LIN {X 0,Y 418.273,Z 271.104,A -85,B 0,C 180,E1 -10135.819,E2 -10135.819} C_VEL
LIN {X 0,Y 422.663,Z 288.535,A -85,B 0,C 180,E1 -10138.973,E2 -10138.973} C_VEL
LIN {X 0,Y 424.828,Z 297.383,A -85,B 0,C 180,E1 -10140.52,E2 -10140.52} C_VEL
LIN {X 0,Y 424.797,Z 302.116,A -85,B 0,C 180,E1 -10141.265,E2 -10141.265} C_VEL
LIN {X 0,Y 423.732,Z 315.882,A -85,B 0,C 180,E1 -10143.326,E2 -10143.326} C_VEL
LIN {X 0,Y 429.33,Z 349.112,A -85,B 0,C 180,E1 -10144.378,E2 -10144.378} C_VEL
LIN {X 0,Y 426.147,Z 475.897,A -85,B 0,C 180,E1 -10146.942,E2 -10146.942} C_VEL
LIN {X 0,Y 425.571,Z 491.648,A -85,B 0,C 180,E1 -10147.359,E2 -10147.359} C_VEL
LIN {X 0,Y 424.744,Z 507.01,A -85,B 0,C 180,E1 -10147.955,E2 -10147.955} C_VEL
LIN {X 0,Y 423.794,Z 521.926,A -85,B 0,C 180,E1 -10148.732,E2 -10148.732} C_VEL
LIN {X 0,Y 422.751,Z 536.416,A -85,B 0,C 180,E1 -10149.696,E2 -10149.696} C_VEL
LIN {X 0,Y 421.703,Z 549.683,A -85,B 0,C 180,E1 -10150.784,E2 -10150.784} C_VEL
LIN {X 0,Y 420.781,Z 561.783,A -85,B 0,C 180,E1 -10151.981,E2 -10151.981} C_VEL
LIN {X 0,Y 419.884,Z 572.417,A -85,B 0,C 180,E1 -10153.22,E2 -10153.22} C_VEL
LIN {X 0,Y 419.045,Z 583.025,A -85,B 0,C 180,E1 -10154.685,E2 -10154.685} C_VEL
LIN {X 0,Y 418.331,Z 593.403,A -85,B 0,C 180,E1 -10156.398,E2 -10156.398} C_VEL
LIN {X 0,Y 417.855,Z 601.99,A -85,B 0,C 180,E1 -10158.111,E2 -10158.111} C_VEL
LIN {X 0,Y 417.459,Z 609.054,A -85,B 0,C 180,E1 -10159.82,E2 -10159.82} C_VEL
LIN {X 0,Y 417.247,Z 615.562,A -85,B 0,C 180,E1 -10161.77,E2 -10161.77} C_VEL
LIN {X 0,Y 417.123,Z 620.649,A -85,B 0,C 180,E1 -10163.763,E2 -10163.763} C_VEL
LIN {X 0,Y 417.095,Z 623.363,A -85,B 0,C 180,E1 -10165.169,E2 -10165.169} C_VEL
LIN {X 0,Y 417.171,Z 625.963,A -85,B 0,C 180,E1 -10167.104,E2 -10167.104} C_VEL
LIN {X 0,Y 417.117,Z 627.235,A -85,B 0,C 180,E1 -10169.036,E2 -10169.036} C_VEL
LIN {X 0,Y 417.106,Z 627.238,A -85,B 0,C 180,E1 -10170.967,E2 -10170.967} C_VEL
LIN {X 0,Y 417.167,Z 625.984,A -85,B 0,C 180,E1 -10172.898,E2 -10172.898} C_VEL
LIN {X 0,Y 417.113,Z 623.451,A -85,B 0,C 180,E1 -10174.834,E2 -10174.834} C_VEL
LIN {X 0,Y 417.146,Z 619.609,A -85,B 0,C 180,E1 -10176.774,E2 -10176.774} C_VEL
LIN {X 0,Y 417.27,Z 614.36,A -85,B 0,C 180,E1 -10178.72,E2 -10178.72} C_VEL
LIN {X 0,Y 417.572,Z 607.571,A -85,B 0,C 180,E1 -10180.67,E2 -10180.67} C_VEL
LIN {X 0,Y 417.913,Z 600.256,A -85,B 0,C 180,E1 -10182.382,E2 -10182.382} C_VEL
LIN {X 0,Y 418.554,Z 591.444,A -85,B 0,C 180,E1 -10184.093,E2 -10184.093} C_VEL
LIN {X 0,Y 419.389,Z 580.845,A -85,B 0,C 180,E1 -10185.803,E2 -10185.803} C_VEL
LIN {X 0,Y 420.33,Z 569.042,A -85,B 0,C 180,E1 -10187.391,E2 -10187.391} C_VEL
LIN {X 0,Y 421.444,Z 557.196,A -85,B 0,C 180,E1 -10188.725,E2 -10188.725} C_VEL
LIN {X 0,Y 422.596,Z 544.432,A -85,B 0,C 180,E1 -10189.934,E2 -10189.934} C_VEL
LIN {X 0,Y 423.78,Z 530.617,A -85,B 0,C 180,E1 -10191.017,E2 -10191.017} C_VEL
LIN {X 0,Y 424.991,Z 515.84,A -85,B 0,C 180,E1 -10191.956,E2 -10191.956} C_VEL
LIN {X 0,Y 426.146,Z 500.139,A -85,B 0,C 180,E1 -10192.733,E2 -10192.733} C_VEL
LIN {X 0,Y 427.209,Z 483.991,A -85,B 0,C 180,E1 -10193.32,E2 -10193.32} C_VEL
LIN {X 0,Y 428.073,Z 463.838,A -85,B 0,C 180,E1 -10193.815,E2 -10193.815} C_VEL
LIN {X 0,Y 431.123,Z 384.555,A -85,B 0,C 180,E1 -10195.656,E2 -10195.656} C_VEL
LIN {X 0,Y 432.678,Z 349.283,A -85,B 0,C 180,E1 -10196.531,E2 -10196.531} C_VEL
LIN {X 0,Y 430.547,Z 332.583,A -85,B 0,C 180,E1 -10197.238,E2 -10197.238} C_VEL
LIN {X 0,Y 427.37,Z 315.726,A -85,B 0,C 180,E1 -10198.1,E2 -10198.1} C_VEL
LIN {X 0,Y 425.847,Z 308.551,A -85,B 0,C 180,E1 -10198.531,E2 -10198.531} C_VEL
LIN {X 0,Y 426.669,Z 302.236,A -85,B 0,C 180,E1 -10199.615,E2 -10199.615} C_VEL
LIN {X 0,Y 425.498,Z 295.343,A -85,B 0,C 180,E1 -10201.076,E2 -10201.076} C_VEL
LIN {X 0,Y 423.264,Z 286.408,A -85,B 0,C 180,E1 -10203.227,E2 -10203.227} C_VEL
LIN {X 0,Y 420.793,Z 278.456,A -85,B 0,C 180,E1 -10205.474,E2 -10205.474} C_VEL
LIN {X 0,Y 418.246,Z 271.014,A -85,B 0,C 180,E1 -10208.054,E2 -10208.054} C_VEL
LIN {X 0,Y 418.229,Z 271.016,A -85,B 0,C 180,E1 -10210.948,E2 -10210.948} C_VEL
LIN {X 0,Y 418.216,Z 271.017,A -85,B 0,C 180,E1 -10213.73,E2 -10213.73} C_VEL
LIN {X 0,Y 418.216,Z 271.016,A -85,B 0,C 180,E1 -10216.449,E2 -10216.449} C_VEL
LIN {X 0,Y 418.229,Z 271.015,A -85,B 0,C 180,E1 -10219.131,E2 -10219.131} C_VEL
LIN {X 0,Y 418.233,Z 271.014,A -85,B 0,C 180,E1 -10222.167,E2 -10222.167} C_VEL
LIN {X 0,Y 418.272,Z 271.011,A -85,B 0,C 180,E1 -10225.42,E2 -10225.42} C_VEL
LIN {X 0,Y 418.236,Z 271.089,A -85,B 0,C 180,E1 -10227.898,E2 -10227.898} C_VEL
LIN {X 0,Y 420.645,Z 278.367,A -85,B 0,C 180,E1 -10230.749,E2 -10230.749} C_VEL
LIN {X 0,Y 420.932,Z 279.274,A -85,B 0,C 180,E1 -10231.015,E2 -10231.015} C_VEL
LIN {X 0,Y 426.506,Z 288.448,A -85,B 0,C 180,E1 -10232.033,E2 -10232.033} C_VEL
LIN {X 0,Y 431.738,Z 298.009,A -85,B 0,C 180,E1 -10232.929,E2 -10232.929} C_VEL
LIN {X 0,Y 434.186,Z 303.111,A -85,B 0,C 180,E1 -10233.341,E2 -10233.341} C_VEL
LIN {X 0,Y 430.286,Z 382.983,A -85,B 0,C 180,E1 -10235.321,E2 -10235.321} C_VEL
LIN {X 0,Y 428.073,Z 441.208,A -85,B 0,C 180,E1 -10236.698,E2 -10236.698} C_VEL
LIN {X 0,Y 427.292,Z 456.973,A -85,B 0,C 180,E1 -10237.262,E2 -10237.262} C_VEL
LIN {X 0,Y 426.378,Z 472.657,A -85,B 0,C 180,E1 -10238.039,E2 -10238.039} C_VEL
LIN {X 0,Y 425.436,Z 486.789,A -85,B 0,C 180,E1 -10238.942,E2 -10238.942} C_VEL
LIN {X 0,Y 424.349,Z 500.509,A -85,B 0,C 180,E1 -10240.026,E2 -10240.026} C_VEL
LIN {X 0,Y 423.148,Z 512.964,A -85,B 0,C 180,E1 -10241.212,E2 -10241.212} C_VEL
LIN {X 0,Y 422.024,Z 524.671,A -85,B 0,C 180,E1 -10242.556,E2 -10242.556} C_VEL
LIN {X 0,Y 421.067,Z 535.277,A -85,B 0,C 180,E1 -10244.013,E2 -10244.013} C_VEL
LIN {X 0,Y 419.97,Z 545.744,A -85,B 0,C 180,E1 -10245.734,E2 -10245.734} C_VEL
LIN {X 0,Y 419.183,Z 554.155,A -85,B 0,C 180,E1 -10247.41,E2 -10247.41} C_VEL
LIN {X 0,Y 418.633,Z 560.313,A -85,B 0,C 180,E1 -10248.868,E2 -10248.868} C_VEL
LIN {X 0,Y 418.092,Z 567.004,A -85,B 0,C 180,E1 -10250.81,E2 -10250.81} C_VEL
LIN {X 0,Y 417.678,Z 572.295,A -85,B 0,C 180,E1 -10252.798,E2 -10252.798} C_VEL
LIN {X 0,Y 417.441,Z 575.139,A -85,B 0,C 180,E1 -10254.202,E2 -10254.202} C_VEL
LIN {X 0,Y 417.373,Z 577.965,A -85,B 0,C 180,E1 -10256.137,E2 -10256.137} C_VEL
LIN {X 0,Y 417.231,Z 579.565,A -85,B 0,C 180,E1 -10258.069,E2 -10258.069} C_VEL
LIN {X 0,Y 417.12,Z 579.956,A -85,B 0,C 180,E1 -10259.999,E2 -10259.999} C_VEL
LIN {X 0,Y 417.179,Z 579.128,A -85,B 0,C 180,E1 -10261.93,E2 -10261.93} C_VEL
LIN {X 0,Y 417.263,Z 577.05,A -85,B 0,C 180,E1 -10263.862,E2 -10263.862} C_VEL
LIN {X 0,Y 417.383,Z 573.711,A -85,B 0,C 180,E1 -10265.798,E2 -10265.798} C_VEL
LIN {X 0,Y 417.568,Z 569.044,A -85,B 0,C 180,E1 -10267.737,E2 -10267.737} C_VEL
LIN {X 0,Y 417.904,Z 562.933,A -85,B 0,C 180,E1 -10269.681,E2 -10269.681} C_VEL
LIN {X 0,Y 418.46,Z 555.198,A -85,B 0,C 180,E1 -10271.626,E2 -10271.626} C_VEL
LIN {X 0,Y 419.056,Z 546.461,A -85,B 0,C 180,E1 -10273.411,E2 -10273.411} C_VEL
LIN {X 0,Y 419.798,Z 536.838,A -85,B 0,C 180,E1 -10275.039,E2 -10275.039} C_VEL
LIN {X 0,Y 420.628,Z 526.543,A -85,B 0,C 180,E1 -10276.501,E2 -10276.501} C_VEL
LIN {X 0,Y 421.633,Z 514.5,A -85,B 0,C 180,E1 -10277.934,E2 -10277.934} C_VEL
LIN {X 0,Y 422.485,Z 501.996,A -85,B 0,C 180,E1 -10279.179,E2 -10279.179} C_VEL
LIN {X 0,Y 423.522,Z 488.72,A -85,B 0,C 180,E1 -10280.266,E2 -10280.266} C_VEL
LIN {X 0,Y 424.403,Z 474.164,A -85,B 0,C 180,E1 -10281.237,E2 -10281.237} C_VEL
LIN {X 0,Y 425.216,Z 459.835,A -85,B 0,C 180,E1 -10281.985,E2 -10281.985} C_VEL
LIN {X 0,Y 425.821,Z 444.87,A -85,B 0,C 180,E1 -10282.579,E2 -10282.579} C_VEL
LIN {X 0,Y 426.282,Z 429.156,A -85,B 0,C 180,E1 -10283.007,E2 -10283.007} C_VEL
LIN {X 0,Y 429.565,Z 298.762,A -85,B 0,C 180,E1 -10285.643,E2 -10285.643} C_VEL
LIN {X 0,Y 420.488,Z 276.554,A -85,B 0,C 180,E1 -10286.661,E2 -10286.661} C_VEL
LIN {X 0,Y 418.28,Z 271.31,A -85,B 0,C 180,E1 -10286.912,E2 -10286.912} C_VEL
LIN {X 0,Y 418.245,Z 271.009,A -85,B 0,C 180,E1 -10286.98,E2 -10286.98} C_VEL
LIN {X 0,Y 418.243,Z 271.013,A -85,B 0,C 180,E1 -10290.271,E2 -10290.271} C_VEL
LIN {X 0,Y 418.249,Z 271.012,A -85,B 0,C 180,E1 -10293.676,E2 -10293.676} C_VEL
LIN {X 0,Y 418.238,Z 271.009,A -85,B 0,C 180,E1 -10297.223,E2 -10297.223} C_VEL
LIN {X 0,Y 418.228,Z 271.015,A -85,B 0,C 180,E1 -10299.683,E2 -10299.683} C_VEL
LIN {X 0,Y 418.222,Z 271.012,A -85,B 0,C 180,E1 -10302.319,E2 -10302.319} C_VEL
LIN {X 0,Y 418.234,Z 271.009,A -85,B 0,C 180,E1 -10305.107,E2 -10305.107} C_VEL
LIN {X 0,Y 418.238,Z 271.015,A -85,B 0,C 180,E1 -10307.765,E2 -10307.765} C_VEL
LIN {X 0,Y 418.243,Z 271.008,A -85,B 0,C 180,E1 -10310.619,E2 -10310.619} C_VEL
LIN {X 0,Y 418.239,Z 271.013,A -85,B 0,C 180,E1 -10313.974,E2 -10313.974} C_VEL
LIN {X 0,Y 418.253,Z 271.008,A -85,B 0,C 180,E1 -10317.155,E2 -10317.155} C_VEL
LIN {X 0,Y 418.257,Z 271.006,A -85,B 0,C 180,E1 -10320.836,E2 -10320.836} C_VEL
LIN {X 0,Y 418.233,Z 271.012,A -85,B 0,C 180,E1 -10324.092,E2 -10324.092} C_VEL
LIN {X 0,Y 418.227,Z 271.012,A -85,B 0,C 180,E1 -10327.262,E2 -10327.262} C_VEL
LIN {X 0,Y 418.277,Z 271.004,A -85,B 0,C 180,E1 -10330.363,E2 -10330.363} C_VEL
LIN {X 0,Y 418.31,Z 271.004,A -85,B 0,C 180,E1 -10333.403,E2 -10333.403} C_VEL
LIN {X 0,Y 418.34,Z 270.996,A -85,B 0,C 180,E1 -10336.998,E2 -10336.998} C_VEL
LIN {X 0,Y 418.315,Z 270.999,A -85,B 0,C 180,E1 -10339.744,E2 -10339.744} C_VEL
LIN {X 0,Y 417.662,Z 271.081,A -85,B 0,C 180,E1 -10340.548,E2 -10340.548} C_VEL
LIN {X 0,Y 414.856,Z 271.434,A -85,B 0,C 180,E1 -10341.857,E2 -10341.857} C_VEL
LIN {X 0,Y 412.502,Z 271.724,A -85,B 0,C 180,E1 -10342.914,E2 -10342.914} C_VEL
LIN {X 0,Y 411.52,Z 271.851,A -85,B 0,C 180,E1 -10343.73,E2 -10343.73} C_VEL
LIN {X 0,Y 411.456,Z 271.854,A -85,B 0,C 180,E1 -10344.006,E2 -10344.006} C_VEL
LIN {X 0,Y 411.502,Z 271.849,A -85,B 0,C 180,E1 -10348.041,E2 -10348.041} C_VEL
LIN {X 0,Y 411.633,Z 271.833,A -85,B 0,C 180,E1 -10349.999,E2 -10349.999} C_VEL
LIN {X 0,Y 411.449,Z 271.855,A -85,B 0,C 180,E1 -10352.936,E2 -10352.936} C_VEL
LIN {X 0,Y 411.448,Z 271.855,A -85,B 0,C 180,E1 -10356.866,E2 -10356.866} C_VEL
LIN {X 0,Y 411.344,Z 271.868,A -85,B 0,C 180,E1 -10358.844,E2 -10358.844} C_VEL
LIN {X 0,Y 411.273,Z 271.879,A -85,B 0,C 180,E1 -10361.832,E2 -10361.832} C_VEL
LIN {X 0,Y 411.249,Z 271.88,A -85,B 0,C 180,E1 -10364.852,E2 -10364.852} C_VEL
LIN {X 0,Y 411.241,Z 271.882,A -85,B 0,C 180,E1 -10367.914,E2 -10367.914} C_VEL
LIN {X 0,Y 411.184,Z 271.89,A -85,B 0,C 180,E1 -10371.033,E2 -10371.033} C_VEL
LIN {X 0,Y 411.213,Z 271.884,A -85,B 0,C 180,E1 -10374.214,E2 -10374.214} C_VEL
LIN {X 0,Y 411.246,Z 271.886,A -85,B 0,C 180,E1 -10377.477,E2 -10377.477} C_VEL
LIN {X 0,Y 411.176,Z 271.89,A -85,B 0,C 180,E1 -10380.847,E2 -10380.847} C_VEL
LIN {X 0,Y 411.192,Z 271.886,A -85,B 0,C 180,E1 -10384.333,E2 -10384.333} C_VEL
LIN {X 0,Y 411.186,Z 271.888,A -85,B 0,C 180,E1 -10387.972,E2 -10387.972} C_VEL
LIN {X 0,Y 411.151,Z 271.898,A -85,B 0,C 180,E1 -10391.228,E2 -10391.228} C_VEL
LIN {X 0,Y 411.167,Z 271.889,A -85,B 0,C 180,E1 -10394.489,E2 -10394.489} C_VEL
LIN {X 0,Y 411.164,Z 271.889,A -85,B 0,C 180,E1 -10398.194,E2 -10398.194} C_VEL
LIN {X 0,Y 411.202,Z 271.887,A -85,B 0,C 180,E1 -10400.776,E2 -10400.776} C_VEL
LIN {X 0,Y 411.183,Z 271.887,A -85,B 0,C 180,E1 -10404.471,E2 -10404.471} C_VEL
LIN {X 0,Y 411.192,Z 271.889,A -85,B 0,C 180,E1 -10406.873,E2 -10406.873} C_VEL
LIN {X 0,Y 411.218,Z 271.884,A -85,B 0,C 180,E1 -10410.644,E2 -10410.644} C_VEL
LIN {X 0,Y 411.223,Z 271.884,A -85,B 0,C 180,E1 -10413.619,E2 -10413.619} C_VEL
LIN {X 0,Y 411.182,Z 271.891,A -85,B 0,C 180,E1 -10416.852,E2 -10416.852} C_VEL
LIN {X 0,Y 411.2,Z 271.885,A -85,B 0,C 180,E1 -10420.051,E2 -10420.051} C_VEL
LIN {X 0,Y 411.249,Z 271.886,A -85,B 0,C 180,E1 -10423.131,E2 -10423.131} C_VEL
LIN {X 0,Y 411.291,Z 271.878,A -85,B 0,C 180,E1 -10426.896,E2 -10426.896} C_VEL
LIN {X 0,Y 411.279,Z 271.875,A -85,B 0,C 180,E1 -10430.162,E2 -10430.162} C_VEL
LIN {X 0,Y 411.438,Z 271.862,A -85,B 0,C 180,E1 -10433.133,E2 -10433.133} C_VEL
LIN {X 0,Y 411.294,Z 271.88,A -85,B 0,C 180,E1 -10435.1,E2 -10435.1} C_VEL
LIN {X 0,Y 411.501,Z 271.847,A -85,B 0,C 180,E1 -10438.043,E2 -10438.043} C_VEL
LIN {X 0,Y 411.628,Z 271.832,A -85,B 0,C 180,E1 -10440.001,E2 -10440.001} C_VEL
LIN {X 0,Y 411.444,Z 271.861,A -85,B 0,C 180,E1 -10442.938,E2 -10442.938} C_VEL
LIN {X 0,Y 411.446,Z 271.86,A -85,B 0,C 180,E1 -10446.868,E2 -10446.868} C_VEL
LIN {X 0,Y 411.342,Z 271.873,A -85,B 0,C 180,E1 -10448.846,E2 -10448.846} C_VEL
LIN {X 0,Y 411.273,Z 271.876,A -85,B 0,C 180,E1 -10451.834,E2 -10451.834} C_VEL
LIN {X 0,Y 411.248,Z 271.885,A -85,B 0,C 180,E1 -10454.854,E2 -10454.854} C_VEL
LIN {X 0,Y 411.241,Z 271.88,A -85,B 0,C 180,E1 -10457.916,E2 -10457.916} C_VEL
LIN {X 0,Y 411.186,Z 271.892,A -85,B 0,C 180,E1 -10461.035,E2 -10461.035} C_VEL
LIN {X 0,Y 411.209,Z 271.885,A -85,B 0,C 180,E1 -10464.217,E2 -10464.217} C_VEL
LIN {X 0,Y 411.249,Z 271.88,A -85,B 0,C 180,E1 -10467.479,E2 -10467.479} C_VEL
LIN {X 0,Y 411.18,Z 271.895,A -85,B 0,C 180,E1 -10470.849,E2 -10470.849} C_VEL
LIN {X 0,Y 411.197,Z 271.887,A -85,B 0,C 180,E1 -10474.335,E2 -10474.335} C_VEL
LIN {X 0,Y 411.184,Z 271.887,A -85,B 0,C 180,E1 -10477.975,E2 -10477.975} C_VEL
LIN {X 0,Y 411.155,Z 271.893,A -85,B 0,C 180,E1 -10481.23,E2 -10481.23} C_VEL
LIN {X 0,Y 411.168,Z 271.893,A -85,B 0,C 180,E1 -10484.492,E2 -10484.492} C_VEL
LIN {X 0,Y 411.171,Z 271.89,A -85,B 0,C 180,E1 -10488.196,E2 -10488.196} C_VEL
LIN {X 0,Y 411.213,Z 271.89,A -85,B 0,C 180,E1 -10490.778,E2 -10490.778} C_VEL
LIN {X 0,Y 411.192,Z 271.888,A -85,B 0,C 180,E1 -10494.473,E2 -10494.473} C_VEL
LIN {X 0,Y 411.24,Z 272.041,A -85,B 0,C 180,E1 -10495.468,E2 -10495.468} C_VEL
LIN {X 0,Y 415.179,Z 287.627,A -85,B 0,C 180,E1 -10498.35,E2 -10498.35} C_VEL
LIN {X 0,Y 418.118,Z 300.046,A -85,B 0,C 180,E1 -10500.553,E2 -10500.553} C_VEL
LIN {X 0,Y 416.971,Z 315.284,A -85,B 0,C 180,E1 -10502.915,E2 -10502.915} C_VEL
LIN {X 0,Y 422.721,Z 350.332,A -85,B 0,C 180,E1 -10504.048,E2 -10504.048} C_VEL
LIN {X 0,Y 419.16,Z 483.298,A -85,B 0,C 180,E1 -10506.829,E2 -10506.829} C_VEL
LIN {X 0,Y 418.407,Z 498.932,A -85,B 0,C 180,E1 -10507.346,E2 -10507.346} C_VEL
LIN {X 0,Y 417.473,Z 513.958,A -85,B 0,C 180,E1 -10508.036,E2 -10508.036} C_VEL
LIN {X 0,Y 416.52,Z 527.842,A -85,B 0,C 180,E1 -10508.861,E2 -10508.861} C_VEL
LIN {X 0,Y 415.547,Z 541.179,A -85,B 0,C 180,E1 -10509.845,E2 -10509.845} C_VEL
LIN {X 0,Y 414.348,Z 554.809,A -85,B 0,C 180,E1 -10511.073,E2 -10511.073} C_VEL
LIN {X 0,Y 413.362,Z 567.287,A -85,B 0,C 180,E1 -10512.437,E2 -10512.437} C_VEL
LIN {X 0,Y 412.381,Z 578.668,A -85,B 0,C 180,E1 -10513.924,E2 -10513.924} C_VEL
LIN {X 0,Y 411.65,Z 588.296,A -85,B 0,C 180,E1 -10515.416,E2 -10515.416} C_VEL
LIN {X 0,Y 410.895,Z 598.331,A -85,B 0,C 180,E1 -10517.29,E2 -10517.29} C_VEL
LIN {X 0,Y 410.529,Z 606.469,A -85,B 0,C 180,E1 -10519.147,E2 -10519.147} C_VEL
LIN {X 0,Y 410.203,Z 613.448,A -85,B 0,C 180,E1 -10521.131,E2 -10521.131} C_VEL
LIN {X 0,Y 410.068,Z 618.866,A -85,B 0,C 180,E1 -10523.111,E2 -10523.111} C_VEL
LIN {X 0,Y 410.024,Z 622.854,A -85,B 0,C 180,E1 -10525.085,E2 -10525.085} C_VEL
LIN {X 0,Y 410.082,Z 625.487,A -85,B 0,C 180,E1 -10527.054,E2 -10527.054} C_VEL
LIN {X 0,Y 410.036,Z 626.789,A -85,B 0,C 180,E1 -10529.019,E2 -10529.019} C_VEL
LIN {X 0,Y 410.026,Z 626.822,A -85,B 0,C 180,E1 -10530.983,E2 -10530.983} C_VEL
LIN {X 0,Y 410.064,Z 625.593,A -85,B 0,C 180,E1 -10532.949,E2 -10532.949} C_VEL
LIN {X 0,Y 410.02,Z 623.081,A -85,B 0,C 180,E1 -10534.918,E2 -10534.918} C_VEL
LIN {X 0,Y 410.054,Z 619.252,A -85,B 0,C 180,E1 -10536.892,E2 -10536.892} C_VEL
LIN {X 0,Y 410.2,Z 614.022,A -85,B 0,C 180,E1 -10538.872,E2 -10538.872} C_VEL
LIN {X 0,Y 410.515,Z 607.248,A -85,B 0,C 180,E1 -10540.856,E2 -10540.856} C_VEL
LIN {X 0,Y 410.927,Z 599.43,A -85,B 0,C 180,E1 -10542.708,E2 -10542.708} C_VEL
LIN {X 0,Y 411.577,Z 591.163,A -85,B 0,C 180,E1 -10544.337,E2 -10544.337} C_VEL
LIN {X 0,Y 412.47,Z 580.62,A -85,B 0,C 180,E1 -10546.075,E2 -10546.075} C_VEL
LIN {X 0,Y 413.508,Z 568.879,A -85,B 0,C 180,E1 -10547.687,E2 -10547.687} C_VEL
LIN {X 0,Y 414.749,Z 555.905,A -85,B 0,C 180,E1 -10549.168,E2 -10549.168} C_VEL
LIN {X 0,Y 416.039,Z 543.023,A -85,B 0,C 180,E1 -10550.391,E2 -10550.391} C_VEL
LIN {X 0,Y 417.3,Z 529.072,A -85,B 0,C 180,E1 -10551.489,E2 -10551.489} C_VEL
LIN {X 0,Y 418.54,Z 515.105,A -85,B 0,C 180,E1 -10552.385,E2 -10552.385} C_VEL
LIN {X 0,Y 419.814,Z 499.081,A -85,B 0,C 180,E1 -10553.187,E2 -10553.187} C_VEL
LIN {X 0,Y 420.954,Z 482.807,A -85,B 0,C 180,E1 -10553.786,E2 -10553.786} C_VEL
LIN {X 0,Y 421.966,Z 459.06,A -85,B 0,C 180,E1 -10554.378,E2 -10554.378} C_VEL
LIN {X 0,Y 425.338,Z 381.047,A -85,B 0,C 180,E1 -10556.26,E2 -10556.26} C_VEL
LIN {X 0,Y 426.828,Z 350.174,A -85,B 0,C 180,E1 -10557.056,E2 -10557.056} C_VEL
LIN {X 0,Y 424.745,Z 333.493,A -85,B 0,C 180,E1 -10557.799,E2 -10557.799} C_VEL
LIN {X 0,Y 421.69,Z 317.064,A -85,B 0,C 180,E1 -10558.69,E2 -10558.69} C_VEL
LIN {X 0,Y 419.738,Z 307.726,A -85,B 0,C 180,E1 -10559.282,E2 -10559.282} C_VEL
LIN {X 0,Y 420.172,Z 304.329,A -85,B 0,C 180,E1 -10559.894,E2 -10559.894} C_VEL
LIN {X 0,Y 419.021,Z 297.809,A -85,B 0,C 180,E1 -10561.33,E2 -10561.33} C_VEL
LIN {X 0,Y 416.858,Z 289.04,A -85,B 0,C 180,E1 -10563.515,E2 -10563.515} C_VEL
LIN {X 0,Y 414.471,Z 281.276,A -85,B 0,C 180,E1 -10565.823,E2 -10565.823} C_VEL
LIN {X 0,Y 412.075,Z 274.472,A -85,B 0,C 180,E1 -10568.322,E2 -10568.322} C_VEL
LIN {X 0,Y 411.232,Z 271.887,A -85,B 0,C 180,E1 -10569.475,E2 -10569.475} C_VEL
LIN {X 0,Y 411.18,Z 271.893,A -85,B 0,C 180,E1 -10573.134,E2 -10573.134} C_VEL
LIN {X 0,Y 411.175,Z 271.894,A -85,B 0,C 180,E1 -10575.881,E2 -10575.881} C_VEL
LIN {X 0,Y 411.17,Z 271.893,A -85,B 0,C 180,E1 -10578.772,E2 -10578.772} C_VEL
LIN {X 0,Y 411.21,Z 271.888,A -85,B 0,C 180,E1 -10581.832,E2 -10581.832} C_VEL
LIN {X 0,Y 411.217,Z 271.889,A -85,B 0,C 180,E1 -10585.122,E2 -10585.122} C_VEL
LIN {X 0,Y 411.241,Z 272.095,A -85,B 0,C 180,E1 -10586.555,E2 -10586.555} C_VEL
LIN {X 0,Y 413.31,Z 278.263,A -85,B 0,C 180,E1 -10589.327,E2 -10589.327} C_VEL
LIN {X 0,Y 413.936,Z 280.267,A -85,B 0,C 180,E1 -10590.085,E2 -10590.085} C_VEL
LIN {X 0,Y 418.128,Z 286.794,A -85,B 0,C 180,E1 -10590.932,E2 -10590.932} C_VEL
LIN {X 0,Y 423.305,Z 295.389,A -85,B 0,C 180,E1 -10591.898,E2 -10591.898} C_VEL
LIN {X 0,Y 428.384,Z 305.503,A -85,B 0,C 180,E1 -10592.817,E2 -10592.817} C_VEL
LIN {X 0,Y 425.343,Z 361.167,A -85,B 0,C 180,E1 -10594.262,E2 -10594.262} C_VEL
LIN {X 0,Y 421.839,Z 442.276,A -85,B 0,C 180,E1 -10596.268,E2 -10596.268} C_VEL
LIN {X 0,Y 420.97,Z 457.94,A -85,B 0,C 180,E1 -10596.845,E2 -10596.845} C_VEL
LIN {X 0,Y 420.002,Z 473.26,A -85,B 0,C 180,E1 -10597.624,E2 -10597.624} C_VEL
LIN {X 0,Y 418.948,Z 488.141,A -85,B 0,C 180,E1 -10598.6,E2 -10598.6} C_VEL
LIN {X 0,Y 417.765,Z 501.665,A -85,B 0,C 180,E1 -10599.697,E2 -10599.697} C_VEL
LIN {X 0,Y 416.413,Z 514.916,A -85,B 0,C 180,E1 -10601,E2 -10601} C_VEL
LIN {X 0,Y 415.304,Z 525.58,A -85,B 0,C 180,E1 -10602.265,E2 -10602.265} C_VEL
LIN {X 0,Y 414.286,Z 536.105,A -85,B 0,C 180,E1 -10603.745,E2 -10603.745} C_VEL
LIN {X 0,Y 413.138,Z 546.503,A -85,B 0,C 180,E1 -10605.493,E2 -10605.493} C_VEL
LIN {X 0,Y 412.26,Z 554.862,A -85,B 0,C 180,E1 -10607.195,E2 -10607.195} C_VEL
LIN {X 0,Y 411.689,Z 560.968,A -85,B 0,C 180,E1 -10608.678,E2 -10608.678} C_VEL
LIN {X 0,Y 411.106,Z 567.619,A -85,B 0,C 180,E1 -10610.653,E2 -10610.653} C_VEL
LIN {X 0,Y 410.655,Z 572.865,A -85,B 0,C 180,E1 -10612.674,E2 -10612.674} C_VEL
LIN {X 0,Y 410.401,Z 575.692,A -85,B 0,C 180,E1 -10614.102,E2 -10614.102} C_VEL
LIN {X 0,Y 410.316,Z 578.473,A -85,B 0,C 180,E1 -10616.071,E2 -10616.071} C_VEL
LIN {X 0,Y 410.155,Z 580.029,A -85,B 0,C 180,E1 -10618.035,E2 -10618.035} C_VEL
LIN {X 0,Y 410.037,Z 580.372,A -85,B 0,C 180,E1 -10619.999,E2 -10619.999} C_VEL
LIN {X 0,Y 410.105,Z 579.493,A -85,B 0,C 180,E1 -10621.963,E2 -10621.963} C_VEL
LIN {X 0,Y 410.171,Z 577.374,A -85,B 0,C 180,E1 -10623.929,E2 -10623.929} C_VEL
LIN {X 0,Y 410.313,Z 573.969,A -85,B 0,C 180,E1 -10625.898,E2 -10625.898} C_VEL
LIN {X 0,Y 410.506,Z 569.229,A -85,B 0,C 180,E1 -10627.871,E2 -10627.871} C_VEL
LIN {X 0,Y 410.851,Z 563.034,A -85,B 0,C 180,E1 -10629.849,E2 -10629.849} C_VEL
LIN {X 0,Y 411.463,Z 555.204,A -85,B 0,C 180,E1 -10631.827,E2 -10631.827} C_VEL
LIN {X 0,Y 412.048,Z 546.902,A -85,B 0,C 180,E1 -10633.537,E2 -10633.537} C_VEL
LIN {X 0,Y 412.879,Z 536.616,A -85,B 0,C 180,E1 -10635.297,E2 -10635.297} C_VEL
LIN {X 0,Y 413.72,Z 526.18,A -85,B 0,C 180,E1 -10636.784,E2 -10636.784} C_VEL
LIN {X 0,Y 414.797,Z 513.811,A -85,B 0,C 180,E1 -10638.259,E2 -10638.259} C_VEL
LIN {X 0,Y 415.716,Z 501.276,A -85,B 0,C 180,E1 -10639.504,E2 -10639.504} C_VEL
LIN {X 0,Y 416.77,Z 487.756,A -85,B 0,C 180,E1 -10640.61,E2 -10640.61} C_VEL
LIN {X 0,Y 417.718,Z 472.872,A -85,B 0,C 180,E1 -10641.594,E2 -10641.594} C_VEL
LIN {X 0,Y 418.554,Z 457.237,A -85,B 0,C 180,E1 -10642.392,E2 -10642.392} C_VEL
LIN {X 0,Y 419.172,Z 441.748,A -85,B 0,C 180,E1 -10642.975,E2 -10642.975} C_VEL
LIN {X 0,Y 419.658,Z 424.509,A -85,B 0,C 180,E1 -10643.403,E2 -10643.403} C_VEL
LIN {X 0,Y 422.929,Z 300.435,A -85,B 0,C 180,E1 -10645.974,E2 -10645.974} C_VEL
LIN {X 0,Y 414.498,Z 279.848,A -85,B 0,C 180,E1 -10646.935,E2 -10646.935} C_VEL
LIN {X 0,Y 411.277,Z 272.478,A -85,B 0,C 180,E1 -10647.302,E2 -10647.302} C_VEL
LIN {X 0,Y 411.202,Z 271.887,A -85,B 0,C 180,E1 -10647.329,E2 -10647.329} C_VEL
LIN {X 0,Y 411.199,Z 271.891,A -85,B 0,C 180,E1 -10649.712,E2 -10649.712} C_VEL
LIN {X 0,Y 411.207,Z 271.884,A -85,B 0,C 180,E1 -10653.154,E2 -10653.154} C_VEL
LIN {X 0,Y 411.192,Z 271.887,A -85,B 0,C 180,E1 -10656.551,E2 -10656.551} C_VEL
LIN {X 0,Y 411.194,Z 271.891,A -85,B 0,C 180,E1 -10659.723,E2 -10659.723} C_VEL
LIN {X 0,Y 411.17,Z 271.889,A -85,B 0,C 180,E1 -10663.133,E2 -10663.133} C_VEL
LIN {X 0,Y 411.166,Z 271.896,A -85,B 0,C 180,E1 -10665.88,E2 -10665.88} C_VEL
LIN {X 0,Y 411.161,Z 271.89,A -85,B 0,C 180,E1 -10668.77,E2 -10668.77} C_VEL
LIN {X 0,Y 411.189,Z 271.891,A -85,B 0,C 180,E1 -10672.024,E2 -10672.024} C_VEL
LIN {X 0,Y 411.202,Z 271.891,A -85,B 0,C 180,E1 -10675.665,E2 -10675.665} C_VEL
LIN {X 0,Y 411.185,Z 271.888,A -85,B 0,C 180,E1 -10679.151,E2 -10679.151} C_VEL
LIN {X 0,Y 411.185,Z 271.887,A -85,B 0,C 180,E1 -10682.516,E2 -10682.516} C_VEL
LIN {X 0,Y 411.207,Z 271.89,A -85,B 0,C 180,E1 -10685.782,E2 -10685.782} C_VEL
LIN {X 0,Y 411.191,Z 271.887,A -85,B 0,C 180,E1 -10688.964,E2 -10688.964} C_VEL
LIN {X 0,Y 411.24,Z 271.882,A -85,B 0,C 180,E1 -10692.083,E2 -10692.083} C_VEL
LIN {X 0,Y 411.253,Z 271.88,A -85,B 0,C 180,E1 -10695.146,E2 -10695.146} C_VEL
LIN {X 0,Y 411.277,Z 271.877,A -85,B 0,C 180,E1 -10698.166,E2 -10698.166} C_VEL
LIN {X 0,Y 411.475,Z 271.852,A -85,B 0,C 180,E1 -10702.145,E2 -10702.145} C_VEL
LIN {X 0,Y 411.456,Z 271.854,A -85,B 0,C 180,E1 -10704.006,E2 -10704.006} C_VEL
LIN {X 0,Y 410.84,Z 271.934,A -85,B 0,C 180,E1 -10704.822,E2 -10704.822} C_VEL
LIN {X 0,Y 408.032,Z 272.286,A -85,B 0,C 180,E1 -10706.149,E2 -10706.149} C_VEL
LIN {X 0,Y 405.609,Z 272.586,A -85,B 0,C 180,E1 -10707.22,E2 -10707.22} C_VEL
LIN {X 0,Y 404.541,Z 272.717,A -85,B 0,C 180,E1 -10708.048,E2 -10708.048} C_VEL
LIN {X 0,Y 404.44,Z 272.727,A -85,B 0,C 180,E1 -10708.329,E2 -10708.329} C_VEL
LIN {X 0,Y 404.602,Z 272.709,A -85,B 0,C 180,E1 -10709.999,E2 -10709.999} C_VEL
LIN {X 0,Y 404.407,Z 272.733,A -85,B 0,C 180,E1 -10712.987,E2 -10712.987} C_VEL
LIN {X 0,Y 404.4,Z 272.734,A -85,B 0,C 180,E1 -10716.986,E2 -10716.986} C_VEL
LIN {X 0,Y 404.248,Z 272.753,A -85,B 0,C 180,E1 -10720.01,E2 -10720.01} C_VEL
LIN {X 0,Y 404.256,Z 272.754,A -85,B 0,C 180,E1 -10723.21,E2 -10723.21} C_VEL
LIN {X 0,Y 404.205,Z 272.759,A -85,B 0,C 180,E1 -10727.006,E2 -10727.006} C_VEL
LIN {X 0,Y 404.152,Z 272.763,A -85,B 0,C 180,E1 -10730.351,E2 -10730.351} C_VEL
LIN {X 0,Y 404.156,Z 272.768,A -85,B 0,C 180,E1 -10733.574,E2 -10733.574} C_VEL
LIN {X 0,Y 404.17,Z 272.764,A -85,B 0,C 180,E1 -10735.765,E2 -10735.765} C_VEL
LIN {X 0,Y 404.182,Z 272.76,A -85,B 0,C 180,E1 -10737.999,E2 -10737.999} C_VEL
LIN {X 0,Y 404.126,Z 272.771,A -85,B 0,C 180,E1 -10741.557,E2 -10741.557} C_VEL
LIN {X 0,Y 404.172,Z 272.764,A -85,B 0,C 180,E1 -10745.015,E2 -10745.015} C_VEL
LIN {X 0,Y 404.144,Z 272.765,A -85,B 0,C 180,E1 -10748.756,E2 -10748.756} C_VEL
LIN {X 0,Y 404.11,Z 272.772,A -85,B 0,C 180,E1 -10751.599,E2 -10751.599} C_VEL
LIN {X 0,Y 404.136,Z 272.765,A -85,B 0,C 180,E1 -10754.522,E2 -10754.522} C_VEL
LIN {X 0,Y 404.125,Z 272.773,A -85,B 0,C 180,E1 -10757.296,E2 -10757.296} C_VEL
LIN {X 0,Y 404.154,Z 272.763,A -85,B 0,C 180,E1 -10759.955,E2 -10759.955} C_VEL
LIN {X 0,Y 404.121,Z 272.773,A -85,B 0,C 180,E1 -10763.125,E2 -10763.125} C_VEL
LIN {X 0,Y 404.13,Z 272.766,A -85,B 0,C 180,E1 -10766.188,E2 -10766.188} C_VEL
LIN {X 0,Y 404.131,Z 272.767,A -85,B 0,C 180,E1 -10769.715,E2 -10769.715} C_VEL
LIN {X 0,Y 404.181,Z 272.766,A -85,B 0,C 180,E1 -10773.123,E2 -10773.123} C_VEL
LIN {X 0,Y 404.16,Z 272.767,A -85,B 0,C 180,E1 -10775.334,E2 -10775.334} C_VEL
LIN {X 0,Y 404.124,Z 272.768,A -85,B 0,C 180,E1 -10778.581,E2 -10778.581} C_VEL
LIN {X 0,Y 404.196,Z 272.758,A -85,B 0,C 180,E1 -10781.762,E2 -10781.762} C_VEL
LIN {X 0,Y 404.191,Z 272.763,A -85,B 0,C 180,E1 -10784.882,E2 -10784.882} C_VEL
LIN {X 0,Y 404.242,Z 272.752,A -85,B 0,C 180,E1 -10787.959,E2 -10787.959} C_VEL
LIN {X 0,Y 404.391,Z 272.733,A -85,B 0,C 180,E1 -10792.13,E2 -10792.13} C_VEL
LIN {X 0,Y 404.405,Z 272.731,A -85,B 0,C 180,E1 -10794.016,E2 -10794.016} C_VEL
LIN {X 0,Y 404.47,Z 272.723,A -85,B 0,C 180,E1 -10798.009,E2 -10798.009} C_VEL
LIN {X 0,Y 404.598,Z 272.707,A -85,B 0,C 180,E1 -10800.001,E2 -10800.001} C_VEL
LIN {X 0,Y 404.402,Z 272.739,A -85,B 0,C 180,E1 -10802.989,E2 -10802.989} C_VEL
LIN {X 0,Y 404.397,Z 272.74,A -85,B 0,C 180,E1 -10806.988,E2 -10806.988} C_VEL
LIN {X 0,Y 404.247,Z 272.751,A -85,B 0,C 180,E1 -10810.013,E2 -10810.013} C_VEL
LIN {X 0,Y 404.255,Z 272.754,A -85,B 0,C 180,E1 -10813.212,E2 -10813.212} C_VEL
LIN {X 0,Y 404.205,Z 272.763,A -85,B 0,C 180,E1 -10817.008,E2 -10817.008} C_VEL
LIN {X 0,Y 404.153,Z 272.764,A -85,B 0,C 180,E1 -10820.353,E2 -10820.353} C_VEL
LIN {X 0,Y 404.153,Z 272.763,A -85,B 0,C 180,E1 -10823.576,E2 -10823.576} C_VEL
LIN {X 0,Y 404.173,Z 272.76,A -85,B 0,C 180,E1 -10825.768,E2 -10825.768} C_VEL
LIN {X 0,Y 404.185,Z 272.759,A -85,B 0,C 180,E1 -10828.001,E2 -10828.001} C_VEL
LIN {X 0,Y 404.13,Z 272.766,A -85,B 0,C 180,E1 -10831.559,E2 -10831.559} C_VEL
LIN {X 0,Y 404.176,Z 272.765,A -85,B 0,C 180,E1 -10835.018,E2 -10835.018} C_VEL
LIN {X 0,Y 404.142,Z 272.771,A -85,B 0,C 180,E1 -10838.759,E2 -10838.759} C_VEL
LIN {X 0,Y 404.115,Z 272.768,A -85,B 0,C 180,E1 -10841.601,E2 -10841.601} C_VEL
LIN {X 0,Y 404.138,Z 272.769,A -85,B 0,C 180,E1 -10844.524,E2 -10844.524} C_VEL
LIN {X 0,Y 404.13,Z 272.767,A -85,B 0,C 180,E1 -10847.297,E2 -10847.297} C_VEL
LIN {X 0,Y 404.163,Z 272.765,A -85,B 0,C 180,E1 -10849.957,E2 -10849.957} C_VEL
LIN {X 0,Y 404.13,Z 272.768,A -85,B 0,C 180,E1 -10853.127,E2 -10853.127} C_VEL
LIN {X 0,Y 404.175,Z 272.886,A -85,B 0,C 180,E1 -10855.099,E2 -10855.099} C_VEL
LIN {X 0,Y 408.252,Z 288.968,A -85,B 0,C 180,E1 -10858.123,E2 -10858.123} C_VEL
LIN {X 0,Y 411.118,Z 300.926,A -85,B 0,C 180,E1 -10860.283,E2 -10860.283} C_VEL
LIN {X 0,Y 411.063,Z 305.285,A -85,B 0,C 180,E1 -10860.988,E2 -10860.988} C_VEL
LIN {X 0,Y 410.222,Z 315.062,A -85,B 0,C 180,E1 -10862.518,E2 -10862.518} C_VEL
LIN {X 0,Y 416.11,Z 351.662,A -85,B 0,C 180,E1 -10863.719,E2 -10863.719} C_VEL
LIN {X 0,Y 412.421,Z 482.725,A -85,B 0,C 180,E1 -10866.528,E2 -10866.528} C_VEL
LIN {X 0,Y 411.625,Z 498.388,A -85,B 0,C 180,E1 -10867.052,E2 -10867.052} C_VEL
LIN {X 0,Y 410.658,Z 513.606,A -85,B 0,C 180,E1 -10867.763,E2 -10867.763} C_VEL
LIN {X 0,Y 409.638,Z 527.757,A -85,B 0,C 180,E1 -10868.62,E2 -10868.62} C_VEL
LIN {X 0,Y 408.637,Z 541.036,A -85,B 0,C 180,E1 -10869.62,E2 -10869.62} C_VEL
LIN {X 0,Y 407.408,Z 554.627,A -85,B 0,C 180,E1 -10870.869,E2 -10870.869} C_VEL
LIN {X 0,Y 406.368,Z 567.214,A -85,B 0,C 180,E1 -10872.272,E2 -10872.272} C_VEL
LIN {X 0,Y 405.453,Z 577.598,A -85,B 0,C 180,E1 -10873.642,E2 -10873.642} C_VEL
LIN {X 0,Y 404.654,Z 587.307,A -85,B 0,C 180,E1 -10875.158,E2 -10875.158} C_VEL
LIN {X 0,Y 403.934,Z 597.149,A -85,B 0,C 180,E1 -10876.993,E2 -10876.993} C_VEL
LIN {X 0,Y 403.487,Z 605.735,A -85,B 0,C 180,E1 -10878.955,E2 -10878.955} C_VEL
LIN {X 0,Y 403.125,Z 612.795,A -85,B 0,C 180,E1 -10880.974,E2 -10880.974} C_VEL
LIN {X 0,Y 402.989,Z 618.282,A -85,B 0,C 180,E1 -10882.989,E2 -10882.989} C_VEL
LIN {X 0,Y 402.953,Z 622.326,A -85,B 0,C 180,E1 -10884.999,E2 -10884.999} C_VEL
LIN {X 0,Y 402.997,Z 624.99,A -85,B 0,C 180,E1 -10887.002,E2 -10887.002} C_VEL
LIN {X 0,Y 402.957,Z 626.336,A -85,B 0,C 180,E1 -10889.002,E2 -10889.002} C_VEL
LIN {X 0,Y 402.948,Z 626.406,A -85,B 0,C 180,E1 -10891.001,E2 -10891.001} C_VEL
LIN {X 0,Y 402.962,Z 625.204,A -85,B 0,C 180,E1 -10893.001,E2 -10893.001} C_VEL
LIN {X 0,Y 402.931,Z 622.721,A -85,B 0,C 180,E1 -10895.004,E2 -10895.004} C_VEL
LIN {X 0,Y 402.975,Z 618.913,A -85,B 0,C 180,E1 -10897.014,E2 -10897.014} C_VEL
LIN {X 0,Y 403.121,Z 613.707,A -85,B 0,C 180,E1 -10899.029,E2 -10899.029} C_VEL
LIN {X 0,Y 403.47,Z 606.961,A -85,B 0,C 180,E1 -10901.048,E2 -10901.048} C_VEL
LIN {X 0,Y 403.995,Z 598.513,A -85,B 0,C 180,E1 -10903.072,E2 -10903.072} C_VEL
LIN {X 0,Y 404.751,Z 589.528,A -85,B 0,C 180,E1 -10904.841,E2 -10904.841} C_VEL
LIN {X 0,Y 405.594,Z 580.445,A -85,B 0,C 180,E1 -10906.355,E2 -10906.355} C_VEL
LIN {X 0,Y 406.713,Z 568.808,A -85,B 0,C 180,E1 -10907.991,E2 -10907.991} C_VEL
LIN {X 0,Y 408.026,Z 555.932,A -85,B 0,C 180,E1 -10909.496,E2 -10909.496} C_VEL
LIN {X 0,Y 409.369,Z 543.195,A -85,B 0,C 180,E1 -10910.739,E2 -10910.739} C_VEL
LIN {X 0,Y 410.717,Z 529.456,A -85,B 0,C 180,E1 -10911.851,E2 -10911.851} C_VEL
LIN {X 0,Y 412.118,Z 514.798,A -85,B 0,C 180,E1 -10912.815,E2 -10912.815} C_VEL
LIN {X 0,Y 413.446,Z 498.76,A -85,B 0,C 180,E1 -10913.639,E2 -10913.639} C_VEL
LIN {X 0,Y 414.675,Z 483.011,A -85,B 0,C 180,E1 -10914.235,E2 -10914.235} C_VEL
LIN {X 0,Y 415.67,Z 461.392,A -85,B 0,C 180,E1 -10914.805,E2 -10914.805} C_VEL
LIN {X 0,Y 419.169,Z 387.159,A -85,B 0,C 180,E1 -10916.649,E2 -10916.649} C_VEL
LIN {X 0,Y 421.076,Z 351.403,A -85,B 0,C 180,E1 -10917.598,E2 -10917.598} C_VEL
LIN {X 0,Y 419.146,Z 335.178,A -85,B 0,C 180,E1 -10918.352,E2 -10918.352} C_VEL
LIN {X 0,Y 416.099,Z 317.976,A -85,B 0,C 180,E1 -10919.33,E2 -10919.33} C_VEL
LIN {X 0,Y 413.677,Z 306.942,A -85,B 0,C 180,E1 -10920.085,E2 -10920.085} C_VEL
LIN {X 0,Y 412.57,Z 300.258,A -85,B 0,C 180,E1 -10921.599,E2 -10921.599} C_VEL
LIN {X 0,Y 410.532,Z 291.853,A -85,B 0,C 180,E1 -10923.79,E2 -10923.79} C_VEL
LIN {X 0,Y 408.332,Z 284.682,A -85,B 0,C 180,E1 -10926.007,E2 -10926.007} C_VEL
LIN {X 0,Y 406.422,Z 279.052,A -85,B 0,C 180,E1 -10928.112,E2 -10928.112} C_VEL
LIN {X 0,Y 405.384,Z 275.875,A -85,B 0,C 180,E1 -10929.513,E2 -10929.513} C_VEL
LIN {X 0,Y 404.15,Z 272.769,A -85,B 0,C 180,E1 -10931.279,E2 -10931.279} C_VEL
LIN {X 0,Y 404.152,Z 272.769,A -85,B 0,C 180,E1 -10934.522,E2 -10934.522} C_VEL
LIN {X 0,Y 404.143,Z 272.769,A -85,B 0,C 180,E1 -10937.296,E2 -10937.296} C_VEL
LIN {X 0,Y 404.176,Z 272.764,A -85,B 0,C 180,E1 -10939.956,E2 -10939.956} C_VEL
LIN {X 0,Y 404.142,Z 272.77,A -85,B 0,C 180,E1 -10943.125,E2 -10943.125} C_VEL
LIN {X 0,Y 404.19,Z 272.89,A -85,B 0,C 180,E1 -10944.726,E2 -10944.726} C_VEL
LIN {X 0,Y 405.356,Z 276.442,A -85,B 0,C 180,E1 -10946.764,E2 -10946.764} C_VEL
LIN {X 0,Y 407.141,Z 281.529,A -85,B 0,C 180,E1 -10949.087,E2 -10949.087} C_VEL
LIN {X 0,Y 413.344,Z 290.898,A -85,B 0,C 180,E1 -10950.437,E2 -10950.437} C_VEL
LIN {X 0,Y 417.331,Z 297.568,A -85,B 0,C 180,E1 -10951.238,E2 -10951.238} C_VEL
LIN {X 0,Y 422.16,Z 306.779,A -85,B 0,C 180,E1 -10952.164,E2 -10952.164} C_VEL
LIN {X 0,Y 422.809,Z 308.833,A -85,B 0,C 180,E1 -10952.312,E2 -10952.312} C_VEL
LIN {X 0,Y 417.975,Z 391.183,A -85,B 0,C 180,E1 -10954.477,E2 -10954.477} C_VEL
LIN {X 0,Y 415.676,Z 442.828,A -85,B 0,C 180,E1 -10955.794,E2 -10955.794} C_VEL
LIN {X 0,Y 414.748,Z 458.372,A -85,B 0,C 180,E1 -10956.381,E2 -10956.381} C_VEL
LIN {X 0,Y 413.673,Z 474.079,A -85,B 0,C 180,E1 -10957.196,E2 -10957.196} C_VEL
LIN {X 0,Y 412.632,Z 487.973,A -85,B 0,C 180,E1 -10958.125,E2 -10958.125} C_VEL
LIN {X 0,Y 411.359,Z 501.571,A -85,B 0,C 180,E1 -10959.236,E2 -10959.236} C_VEL
LIN {X 0,Y 409.944,Z 514.794,A -85,B 0,C 180,E1 -10960.548,E2 -10960.548} C_VEL
LIN {X 0,Y 408.61,Z 526.577,A -85,B 0,C 180,E1 -10961.964,E2 -10961.964} C_VEL
LIN {X 0,Y 407.529,Z 537.004,A -85,B 0,C 180,E1 -10963.467,E2 -10963.467} C_VEL
LIN {X 0,Y 406.323,Z 547.324,A -85,B 0,C 180,E1 -10965.244,E2 -10965.244} C_VEL
LIN {X 0,Y 405.349,Z 555.617,A -85,B 0,C 180,E1 -10966.973,E2 -10966.973} C_VEL
LIN {X 0,Y 404.528,Z 563.476,A -85,B 0,C 180,E1 -10968.982,E2 -10968.982} C_VEL
LIN {X 0,Y 403.956,Z 569.678,A -85,B 0,C 180,E1 -10970.991,E2 -10970.991} C_VEL
LIN {X 0,Y 403.556,Z 574.541,A -85,B 0,C 180,E1 -10973.062,E2 -10973.062} C_VEL
LIN {X 0,Y 403.185,Z 577.794,A -85,B 0,C 180,E1 -10974.999,E2 -10974.999} C_VEL
LIN {X 0,Y 403.26,Z 578.993,A -85,B 0,C 180,E1 -10976.002,E2 -10976.002} C_VEL
LIN {X 0,Y 403.081,Z 580.499,A -85,B 0,C 180,E1 -10978.001,E2 -10978.001} C_VEL
LIN {X 0,Y 402.956,Z 580.788,A -85,B 0,C 180,E1 -10979.999,E2 -10979.999} C_VEL
LIN {X 0,Y 403.035,Z 579.848,A -85,B 0,C 180,E1 -10981.998,E2 -10981.998} C_VEL
LIN {X 0,Y 403.131,Z 578.919,A -85,B 0,C 180,E1 -10982.997,E2 -10982.997} C_VEL
LIN {X 0,Y 403.115,Z 576.116,A -85,B 0,C 180,E1 -10985,E2 -10985} C_VEL
LIN {X 0,Y 403.358,Z 571.981,A -85,B 0,C 180,E1 -10987.005,E2 -10987.005} C_VEL
LIN {X 0,Y 403.609,Z 566.45,A -85,B 0,C 180,E1 -10989.015,E2 -10989.015} C_VEL
LIN {X 0,Y 404.042,Z 559.371,A -85,B 0,C 180,E1 -10991.03,E2 -10991.03} C_VEL
LIN {X 0,Y 404.692,Z 551.695,A -85,B 0,C 180,E1 -10992.792,E2 -10992.792} C_VEL
LIN {X 0,Y 405.412,Z 542.445,A -85,B 0,C 180,E1 -10994.557,E2 -10994.557} C_VEL
LIN {X 0,Y 406.255,Z 532.982,A -85,B 0,C 180,E1 -10996.068,E2 -10996.068} C_VEL
LIN {X 0,Y 407.194,Z 521.782,A -85,B 0,C 180,E1 -10997.579,E2 -10997.579} C_VEL
LIN {X 0,Y 408.245,Z 509.417,A -85,B 0,C 180,E1 -10998.973,E2 -10998.973} C_VEL
LIN {X 0,Y 409.308,Z 496.134,A -85,B 0,C 180,E1 -11000.215,E2 -11000.215} C_VEL
LIN {X 0,Y 410.253,Z 483.12,A -85,B 0,C 180,E1 -11001.215,E2 -11001.215} C_VEL
LIN {X 0,Y 411.202,Z 469.12,A -85,B 0,C 180,E1 -11002.086,E2 -11002.086} C_VEL
LIN {X 0,Y 411.955,Z 453.27,A -85,B 0,C 180,E1 -11002.854,E2 -11002.854} C_VEL
LIN {X 0,Y 412.563,Z 438.684,A -85,B 0,C 180,E1 -11003.364,E2 -11003.364} C_VEL
LIN {X 0,Y 413.211,Z 414.279,A -85,B 0,C 180,E1 -11003.924,E2 -11003.924} C_VEL
LIN {X 0,Y 416.354,Z 302.272,A -85,B 0,C 180,E1 -11006.302,E2 -11006.302} C_VEL
LIN {X 0,Y 408.319,Z 282.641,A -85,B 0,C 180,E1 -11007.239,E2 -11007.239} C_VEL
LIN {X 0,Y 404.255,Z 273.369,A -85,B 0,C 180,E1 -11007.711,E2 -11007.711} C_VEL
LIN {X 0,Y 404.134,Z 272.77,A -85,B 0,C 180,E1 -11007.734,E2 -11007.734} C_VEL
LIN {X 0,Y 404.145,Z 272.769,A -85,B 0,C 180,E1 -11010.284,E2 -11010.284} C_VEL
LIN {X 0,Y 404.146,Z 272.77,A -85,B 0,C 180,E1 -11013.811,E2 -11013.811} C_VEL
LIN {X 0,Y 404.134,Z 272.765,A -85,B 0,C 180,E1 -11016.873,E2 -11016.873} C_VEL
LIN {X 0,Y 404.147,Z 272.768,A -85,B 0,C 180,E1 -11020.079,E2 -11020.079} C_VEL
LIN {X 0,Y 404.149,Z 272.764,A -85,B 0,C 180,E1 -11023.082,E2 -11023.082} C_VEL
LIN {X 0,Y 404.146,Z 272.77,A -85,B 0,C 180,E1 -11025.924,E2 -11025.924} C_VEL
LIN {X 0,Y 404.116,Z 272.768,A -85,B 0,C 180,E1 -11028.633,E2 -11028.633} C_VEL
LIN {X 0,Y 404.148,Z 272.767,A -85,B 0,C 180,E1 -11031.491,E2 -11031.491} C_VEL
LIN {X 0,Y 404.18,Z 272.76,A -85,B 0,C 180,E1 -11034.982,E2 -11034.982} C_VEL
LIN {X 0,Y 404.135,Z 272.766,A -85,B 0,C 180,E1 -11038.441,E2 -11038.441} C_VEL
LIN {X 0,Y 404.153,Z 272.763,A -85,B 0,C 180,E1 -11040.861,E2 -11040.861} C_VEL
LIN {X 0,Y 404.146,Z 272.765,A -85,B 0,C 180,E1 -11044.23,E2 -11044.23} C_VEL
LIN {X 0,Y 404.163,Z 272.767,A -85,B 0,C 180,E1 -11047.507,E2 -11047.507} C_VEL
LIN {X 0,Y 404.157,Z 272.762,A -85,B 0,C 180,E1 -11050.706,E2 -11050.706} C_VEL
LIN {X 0,Y 404.215,Z 272.76,A -85,B 0,C 180,E1 -11053.847,E2 -11053.847} C_VEL
LIN {X 0,Y 404.276,Z 272.748,A -85,B 0,C 180,E1 -11056.937,E2 -11056.937} C_VEL
LIN {X 0,Y 404.251,Z 272.754,A -85,B 0,C 180,E1 -11059.987,E2 -11059.987} C_VEL
LIN {X 0,Y 404.402,Z 272.733,A -85,B 0,C 180,E1 -11063.011,E2 -11063.011} C_VEL
LIN {X 0,Y 404.271,Z 272.749,A -85,B 0,C 180,E1 -11065.012,E2 -11065.012} C_VEL
LIN {X 0,Y 404.44,Z 272.727,A -85,B 0,C 180,E1 -11068.329,E2 -11068.329} C_VEL
LIN {X 0,Y 403.743,Z 272.819,A -85,B 0,C 180,E1 -11069.16,E2 -11069.16} C_VEL
LIN {X 0,Y 400.901,Z 273.168,A -85,B 0,C 180,E1 -11070.511,E2 -11070.511} C_VEL
LIN {X 0,Y 398.508,Z 273.473,A -85,B 0,C 180,E1 -11071.603,E2 -11071.603} C_VEL
LIN {X 0,Y 397.468,Z 273.596,A -85,B 0,C 180,E1 -11072.446,E2 -11072.446} C_VEL
LIN {X 0,Y 397.376,Z 273.607,A -85,B 0,C 180,E1 -11072.732,E2 -11072.732} C_VEL
LIN {X 0,Y 397.363,Z 273.61,A -85,B 0,C 180,E1 -11076.09,E2 -11076.09} C_VEL
LIN {X 0,Y 397.368,Z 273.609,A -85,B 0,C 180,E1 -11078.133,E2 -11078.133} C_VEL
LIN {X 0,Y 397.209,Z 273.628,A -85,B 0,C 180,E1 -11082.257,E2 -11082.257} C_VEL
LIN {X 0,Y 397.168,Z 273.639,A -85,B 0,C 180,E1 -11085.391,E2 -11085.391} C_VEL
LIN {X 0,Y 397.15,Z 273.635,A -85,B 0,C 180,E1 -11088.572,E2 -11088.572} C_VEL
LIN {X 0,Y 397.096,Z 273.645,A -85,B 0,C 180,E1 -11091.817,E2 -11091.817} C_VEL
LIN {X 0,Y 397.14,Z 273.642,A -85,B 0,C 180,E1 -11095.511,E2 -11095.511} C_VEL
LIN {X 0,Y 397.109,Z 273.641,A -85,B 0,C 180,E1 -11098.543,E2 -11098.543} C_VEL
LIN {X 0,Y 397.065,Z 273.646,A -85,B 0,C 180,E1 -11102.071,E2 -11102.071} C_VEL
LIN {X 0,Y 397.106,Z 273.646,A -85,B 0,C 180,E1 -11105.503,E2 -11105.503} C_VEL
LIN {X 0,Y 397.119,Z 273.641,A -85,B 0,C 180,E1 -11108.861,E2 -11108.861} C_VEL
LIN {X 0,Y 397.056,Z 273.647,A -85,B 0,C 180,E1 -11112.266,E2 -11112.266} C_VEL
LIN {X 0,Y 397.078,Z 273.649,A -85,B 0,C 180,E1 -11115.068,E2 -11115.068} C_VEL
LIN {X 0,Y 397.053,Z 273.648,A -85,B 0,C 180,E1 -11118.02,E2 -11118.02} C_VEL
LIN {X 0,Y 397.115,Z 273.645,A -85,B 0,C 180,E1 -11121.138,E2 -11121.138} C_VEL
LIN {X 0,Y 397.105,Z 273.641,A -85,B 0,C 180,E1 -11124.496,E2 -11124.496} C_VEL
LIN {X 0,Y 397.063,Z 273.647,A -85,B 0,C 180,E1 -11127.928,E2 -11127.928} C_VEL
LIN {X 0,Y 397.107,Z 273.644,A -85,B 0,C 180,E1 -11131.456,E2 -11131.456} C_VEL
LIN {X 0,Y 397.138,Z 273.637,A -85,B 0,C 180,E1 -11134.488,E2 -11134.488} C_VEL
LIN {X 0,Y 397.081,Z 273.644,A -85,B 0,C 180,E1 -11138.182,E2 -11138.182} C_VEL
LIN {X 0,Y 397.148,Z 273.639,A -85,B 0,C 180,E1 -11141.427,E2 -11141.427} C_VEL
LIN {X 0,Y 397.164,Z 273.635,A -85,B 0,C 180,E1 -11144.608,E2 -11144.608} C_VEL
LIN {X 0,Y 397.205,Z 273.629,A -85,B 0,C 180,E1 -11147.742,E2 -11147.742} C_VEL
LIN {X 0,Y 397.239,Z 273.628,A -85,B 0,C 180,E1 -11150.839,E2 -11150.839} C_VEL
LIN {X 0,Y 397.356,Z 273.61,A -85,B 0,C 180,E1 -11153.909,E2 -11153.909} C_VEL
LIN {X 0,Y 397.439,Z 273.599,A -85,B 0,C 180,E1 -11157.974,E2 -11157.974} C_VEL
LIN {X 0,Y 397.567,Z 273.583,A -85,B 0,C 180,E1 -11160.001,E2 -11160.001} C_VEL
LIN {X 0,Y 397.362,Z 273.616,A -85,B 0,C 180,E1 -11163.042,E2 -11163.042} C_VEL
LIN {X 0,Y 397.35,Z 273.616,A -85,B 0,C 180,E1 -11167.113,E2 -11167.113} C_VEL
LIN {X 0,Y 397.206,Z 273.629,A -85,B 0,C 180,E1 -11170.192,E2 -11170.192} C_VEL
LIN {X 0,Y 397.215,Z 273.63,A -85,B 0,C 180,E1 -11173.322,E2 -11173.322} C_VEL
LIN {X 0,Y 397.171,Z 273.637,A -85,B 0,C 180,E1 -11177.156,E2 -11177.156} C_VEL
LIN {X 0,Y 397.092,Z 273.648,A -85,B 0,C 180,E1 -11180.731,E2 -11180.731} C_VEL
LIN {X 0,Y 397.118,Z 273.639,A -85,B 0,C 180,E1 -11184.02,E2 -11184.02} C_VEL
LIN {X 0,Y 397.185,Z 273.632,A -85,B 0,C 180,E1 -11187.391,E2 -11187.391} C_VEL
LIN {X 0,Y 397.07,Z 273.652,A -85,B 0,C 180,E1 -11190.884,E2 -11190.884} C_VEL
LIN {X 0,Y 397.116,Z 273.643,A -85,B 0,C 180,E1 -11194.495,E2 -11194.495} C_VEL
LIN {X 0,Y 397.092,Z 273.644,A -85,B 0,C 180,E1 -11198.277,E2 -11198.277} C_VEL
LIN {X 0,Y 397.081,Z 273.649,A -85,B 0,C 180,E1 -11200.91,E2 -11200.91} C_VEL
LIN {X 0,Y 397.093,Z 273.642,A -85,B 0,C 180,E1 -11203.65,E2 -11203.65} C_VEL
LIN {X 0,Y 397.095,Z 273.647,A -85,B 0,C 180,E1 -11206.523,E2 -11206.523} C_VEL
LIN {X 0,Y 397.108,Z 273.647,A -85,B 0,C 180,E1 -11210.424,E2 -11210.424} C_VEL
LIN {X 0,Y 397.102,Z 273.642,A -85,B 0,C 180,E1 -11214.267,E2 -11214.267} C_VEL
LIN {X 0,Y 397.162,Z 273.744,A -85,B 0,C 180,E1 -11214.724,E2 -11214.724} C_VEL
LIN {X 0,Y 401.177,Z 289.742,A -85,B 0,C 180,E1 -11217.79,E2 -11217.79} C_VEL
LIN {X 0,Y 404.216,Z 302.37,A -85,B 0,C 180,E1 -11220.11,E2 -11220.11} C_VEL
LIN {X 0,Y 404.275,Z 305.836,A -85,B 0,C 180,E1 -11220.688,E2 -11220.688} C_VEL
LIN {X 0,Y 403.473,Z 314.719,A -85,B 0,C 180,E1 -11222.104,E2 -11222.104} C_VEL
LIN {X 0,Y 409.499,Z 352.182,A -85,B 0,C 180,E1 -11223.363,E2 -11223.363} C_VEL
LIN {X 0,Y 405.654,Z 481.951,A -85,B 0,C 180,E1 -11226.214,E2 -11226.214} C_VEL
LIN {X 0,Y 404.838,Z 498.108,A -85,B 0,C 180,E1 -11226.766,E2 -11226.766} C_VEL
LIN {X 0,Y 403.828,Z 513.309,A -85,B 0,C 180,E1 -11227.49,E2 -11227.49} C_VEL
LIN {X 0,Y 402.755,Z 527.58,A -85,B 0,C 180,E1 -11228.371,E2 -11228.371} C_VEL
LIN {X 0,Y 401.719,Z 540.822,A -85,B 0,C 180,E1 -11229.387,E2 -11229.387} C_VEL
LIN {X 0,Y 400.453,Z 554.391,A -85,B 0,C 180,E1 -11230.656,E2 -11230.656} C_VEL
LIN {X 0,Y 399.383,Z 566.778,A -85,B 0,C 180,E1 -11232.059,E2 -11232.059} C_VEL
LIN {X 0,Y 398.374,Z 578.191,A -85,B 0,C 180,E1 -11233.606,E2 -11233.606} C_VEL
LIN {X 0,Y 397.55,Z 587.8,A -85,B 0,C 180,E1 -11235.149,E2 -11235.149} C_VEL
LIN {X 0,Y 396.854,Z 596.989,A -85,B 0,C 180,E1 -11236.91,E2 -11236.91} C_VEL
LIN {X 0,Y 396.448,Z 604.96,A -85,B 0,C 180,E1 -11238.757,E2 -11238.757} C_VEL
LIN {X 0,Y 396.037,Z 612.117,A -85,B 0,C 180,E1 -11240.811,E2 -11240.811} C_VEL
LIN {X 0,Y 395.91,Z 617.678,A -85,B 0,C 180,E1 -11242.863,E2 -11242.863} C_VEL
LIN {X 0,Y 395.864,Z 621.77,A -85,B 0,C 180,E1 -11244.909,E2 -11244.909} C_VEL
LIN {X 0,Y 395.898,Z 624.481,A -85,B 0,C 180,E1 -11246.949,E2 -11246.949} C_VEL
LIN {X 0,Y 395.882,Z 625.877,A -85,B 0,C 180,E1 -11248.984,E2 -11248.984} C_VEL
LIN {X 0,Y 395.874,Z 625.99,A -85,B 0,C 180,E1 -11251.019,E2 -11251.019} C_VEL
LIN {X 0,Y 395.861,Z 624.82,A -85,B 0,C 180,E1 -11253.054,E2 -11253.054} C_VEL
LIN {X 0,Y 395.845,Z 622.37,A -85,B 0,C 180,E1 -11255.094,E2 -11255.094} C_VEL
LIN {X 0,Y 395.897,Z 618.597,A -85,B 0,C 180,E1 -11257.14,E2 -11257.14} C_VEL
LIN {X 0,Y 396.033,Z 613.418,A -85,B 0,C 180,E1 -11259.192,E2 -11259.192} C_VEL
LIN {X 0,Y 396.434,Z 606.71,A -85,B 0,C 180,E1 -11261.247,E2 -11261.247} C_VEL
LIN {X 0,Y 397.003,Z 598.302,A -85,B 0,C 180,E1 -11263.306,E2 -11263.306} C_VEL
LIN {X 0,Y 397.817,Z 589.37,A -85,B 0,C 180,E1 -11265.106,E2 -11265.106} C_VEL
LIN {X 0,Y 398.902,Z 578.668,A -85,B 0,C 180,E1 -11266.901,E2 -11266.901} C_VEL
LIN {X 0,Y 400.096,Z 567.603,A -85,B 0,C 180,E1 -11268.458,E2 -11268.458} C_VEL
LIN {X 0,Y 401.315,Z 556.056,A -85,B 0,C 180,E1 -11269.836,E2 -11269.836} C_VEL
LIN {X 0,Y 402.893,Z 542.058,A -85,B 0,C 180,E1 -11271.222,E2 -11271.222} C_VEL
LIN {X 0,Y 404.338,Z 528.263,A -85,B 0,C 180,E1 -11272.349,E2 -11272.349} C_VEL
LIN {X 0,Y 405.78,Z 513.959,A -85,B 0,C 180,E1 -11273.302,E2 -11273.302} C_VEL
LIN {X 0,Y 407.225,Z 497.983,A -85,B 0,C 180,E1 -11274.134,E2 -11274.134} C_VEL
LIN {X 0,Y 408.566,Z 481.73,A -85,B 0,C 180,E1 -11274.757,E2 -11274.757} C_VEL
LIN {X 0,Y 409.718,Z 456.82,A -85,B 0,C 180,E1 -11275.429,E2 -11275.429} C_VEL
LIN {X 0,Y 413.339,Z 388.249,A -85,B 0,C 180,E1 -11277.192,E2 -11277.192} C_VEL
LIN {X 0,Y 415.387,Z 352.315,A -85,B 0,C 180,E1 -11278.184,E2 -11278.184} C_VEL
LIN {X 0,Y 413.754,Z 337.497,A -85,B 0,C 180,E1 -11278.899,E2 -11278.899} C_VEL
LIN {X 0,Y 411.015,Z 321.061,A -85,B 0,C 180,E1 -11279.868,E2 -11279.868} C_VEL
LIN {X 0,Y 408.643,Z 310.338,A -85,B 0,C 180,E1 -11280.63,E2 -11280.63} C_VEL
LIN {X 0,Y 406.803,Z 306.05,A -85,B 0,C 180,E1 -11281.084,E2 -11281.084} C_VEL
LIN {X 0,Y 404.71,Z 296.568,A -85,B 0,C 180,E1 -11283.535,E2 -11283.535} C_VEL
LIN {X 0,Y 402.708,Z 289.553,A -85,B 0,C 180,E1 -11285.692,E2 -11285.692} C_VEL
LIN {X 0,Y 400.758,Z 283.655,A -85,B 0,C 180,E1 -11287.893,E2 -11287.893} C_VEL
LIN {X 0,Y 399.408,Z 279.674,A -85,B 0,C 180,E1 -11289.715,E2 -11289.715} C_VEL
LIN {X 0,Y 398.396,Z 277.108,A -85,B 0,C 180,E1 -11291.184,E2 -11291.184} C_VEL
LIN {X 0,Y 397.116,Z 273.645,A -85,B 0,C 180,E1 -11293.999,E2 -11293.999} C_VEL
LIN {X 0,Y 397.109,Z 273.645,A -85,B 0,C 180,E1 -11296.521,E2 -11296.521} C_VEL
LIN {X 0,Y 397.12,Z 273.644,A -85,B 0,C 180,E1 -11300.423,E2 -11300.423} C_VEL
LIN {X 0,Y 397.109,Z 273.728,A -85,B 0,C 180,E1 -11302.015,E2 -11302.015} C_VEL
LIN {X 0,Y 398.405,Z 277.394,A -85,B 0,C 180,E1 -11305.018,E2 -11305.018} C_VEL
LIN {X 0,Y 400.282,Z 282.728,A -85,B 0,C 180,E1 -11307.94,E2 -11307.94} C_VEL
LIN {X 0,Y 403.18,Z 286.768,A -85,B 0,C 180,E1 -11308.666,E2 -11308.666} C_VEL
LIN {X 0,Y 408.877,Z 295.338,A -85,B 0,C 180,E1 -11309.97,E2 -11309.97} C_VEL
LIN {X 0,Y 414.184,Z 304.552,A -85,B 0,C 180,E1 -11311.092,E2 -11311.092} C_VEL
LIN {X 0,Y 417.233,Z 310.689,A -85,B 0,C 180,E1 -11311.713,E2 -11311.713} C_VEL
LIN {X 0,Y 412.446,Z 385.618,A -85,B 0,C 180,E1 -11313.77,E2 -11313.77} C_VEL
LIN {X 0,Y 409.607,Z 443.174,A -85,B 0,C 180,E1 -11315.287,E2 -11315.287} C_VEL
LIN {X 0,Y 408.64,Z 458.462,A -85,B 0,C 180,E1 -11315.876,E2 -11315.876} C_VEL
LIN {X 0,Y 407.492,Z 474.084,A -85,B 0,C 180,E1 -11316.696,E2 -11316.696} C_VEL
LIN {X 0,Y 406.367,Z 487.989,A -85,B 0,C 180,E1 -11317.636,E2 -11317.636} C_VEL
LIN {X 0,Y 405.009,Z 501.622,A -85,B 0,C 180,E1 -11318.762,E2 -11318.762} C_VEL
LIN {X 0,Y 403.611,Z 514.291,A -85,B 0,C 180,E1 -11320.031,E2 -11320.031} C_VEL
LIN {X 0,Y 402.153,Z 525.75,A -85,B 0,C 180,E1 -11321.401,E2 -11321.401} C_VEL
LIN {X 0,Y 400.987,Z 536.367,A -85,B 0,C 180,E1 -11322.927,E2 -11322.927} C_VEL
LIN {X 0,Y 399.698,Z 546.723,A -85,B 0,C 180,E1 -11324.707,E2 -11324.707} C_VEL
LIN {X 0,Y 398.569,Z 555.315,A -85,B 0,C 180,E1 -11326.488,E2 -11326.488} C_VEL
LIN {X 0,Y 397.828,Z 562.406,A -85,B 0,C 180,E1 -11328.278,E2 -11328.278} C_VEL
LIN {X 0,Y 397.136,Z 568.938,A -85,B 0,C 180,E1 -11330.321,E2 -11330.321} C_VEL
LIN {X 0,Y 396.619,Z 573.976,A -85,B 0,C 180,E1 -11332.362,E2 -11332.362} C_VEL
LIN {X 0,Y 396.329,Z 576.851,A -85,B 0,C 180,E1 -11333.892,E2 -11333.892} C_VEL
LIN {X 0,Y 396.206,Z 579.525,A -85,B 0,C 180,E1 -11335.931,E2 -11335.931} C_VEL
LIN {X 0,Y 396.01,Z 580.977,A -85,B 0,C 180,E1 -11337.965,E2 -11337.965} C_VEL
LIN {X 0,Y 395.878,Z 581.204,A -85,B 0,C 180,E1 -11339.999,E2 -11339.999} C_VEL
LIN {X 0,Y 395.967,Z 580.199,A -85,B 0,C 180,E1 -11342.033,E2 -11342.033} C_VEL
LIN {X 0,Y 395.991,Z 577.969,A -85,B 0,C 180,E1 -11344.07,E2 -11344.07} C_VEL
LIN {X 0,Y 396.183,Z 574.441,A -85,B 0,C 180,E1 -11346.109,E2 -11346.109} C_VEL
LIN {X 0,Y 396.389,Z 569.542,A -85,B 0,C 180,E1 -11348.153,E2 -11348.153} C_VEL
LIN {X 0,Y 396.79,Z 563.16,A -85,B 0,C 180,E1 -11350.201,E2 -11350.201} C_VEL
LIN {X 0,Y 397.373,Z 556.185,A -85,B 0,C 180,E1 -11351.993,E2 -11351.993} C_VEL
LIN {X 0,Y 397.992,Z 547.828,A -85,B 0,C 180,E1 -11353.775,E2 -11353.775} C_VEL
LIN {X 0,Y 398.742,Z 539.139,A -85,B 0,C 180,E1 -11355.329,E2 -11355.329} C_VEL
LIN {X 0,Y 399.649,Z 529.008,A -85,B 0,C 180,E1 -11356.867,E2 -11356.867} C_VEL
LIN {X 0,Y 400.747,Z 516.94,A -85,B 0,C 180,E1 -11358.4,E2 -11358.4} C_VEL
LIN {X 0,Y 401.778,Z 503.602,A -85,B 0,C 180,E1 -11359.81,E2 -11359.81} C_VEL
LIN {X 0,Y 402.901,Z 490.412,A -85,B 0,C 180,E1 -11360.951,E2 -11360.951} C_VEL
LIN {X 0,Y 403.893,Z 476.014,A -85,B 0,C 180,E1 -11361.969,E2 -11361.969} C_VEL
LIN {X 0,Y 404.812,Z 461.126,A -85,B 0,C 180,E1 -11362.795,E2 -11362.795} C_VEL
LIN {X 0,Y 405.506,Z 445.376,A -85,B 0,C 180,E1 -11363.456,E2 -11363.456} C_VEL
LIN {X 0,Y 406.047,Z 429.921,A -85,B 0,C 180,E1 -11363.898,E2 -11363.898} C_VEL
LIN {X 0,Y 409.7,Z 303.894,A -85,B 0,C 180,E1 -11366.644,E2 -11366.644} C_VEL
LIN {X 0,Y 402.335,Z 285.949,A -85,B 0,C 180,E1 -11367.518,E2 -11367.518} C_VEL
LIN {X 0,Y 397.215,Z 274.318,A -85,B 0,C 180,E1 -11368.125,E2 -11368.125} C_VEL
LIN {X 0,Y 397.091,Z 273.647,A -85,B 0,C 180,E1 -11368.182,E2 -11368.182} C_VEL
LIN {X 0,Y 397.079,Z 273.646,A -85,B 0,C 180,E1 -11370.881,E2 -11370.881} C_VEL
LIN {X 0,Y 397.126,Z 273.639,A -85,B 0,C 180,E1 -11374.492,E2 -11374.492} C_VEL
LIN {X 0,Y 397.095,Z 273.645,A -85,B 0,C 180,E1 -11378.274,E2 -11378.274} C_VEL
LIN {X 0,Y 397.061,Z 273.646,A -85,B 0,C 180,E1 -11380.911,E2 -11380.911} C_VEL
LIN {X 0,Y 397.099,Z 273.646,A -85,B 0,C 180,E1 -11383.647,E2 -11383.647} C_VEL
LIN {X 0,Y 397.1,Z 273.642,A -85,B 0,C 180,E1 -11386.52,E2 -11386.52} C_VEL
LIN {X 0,Y 397.11,Z 273.641,A -85,B 0,C 180,E1 -11390.421,E2 -11390.421} C_VEL
LIN {X 0,Y 397.105,Z 273.643,A -85,B 0,C 180,E1 -11394.264,E2 -11394.264} C_VEL
LIN {X 0,Y 397.111,Z 273.64,A -85,B 0,C 180,E1 -11396.726,E2 -11396.726} C_VEL
LIN {X 0,Y 397.114,Z 273.641,A -85,B 0,C 180,E1 -11400.294,E2 -11400.294} C_VEL
LIN {X 0,Y 397.091,Z 273.65,A -85,B 0,C 180,E1 -11403.737,E2 -11403.737} C_VEL
LIN {X 0,Y 397.099,Z 273.643,A -85,B 0,C 180,E1 -11407.084,E2 -11407.084} C_VEL
LIN {X 0,Y 397.141,Z 273.637,A -85,B 0,C 180,E1 -11410.351,E2 -11410.351} C_VEL
LIN {X 0,Y 397.16,Z 273.64,A -85,B 0,C 180,E1 -11413.552,E2 -11413.552} C_VEL
LIN {X 0,Y 397.223,Z 273.626,A -85,B 0,C 180,E1 -11416.701,E2 -11416.701} C_VEL
LIN {X 0,Y 397.211,Z 273.632,A -85,B 0,C 180,E1 -11419.808,E2 -11419.808} C_VEL
LIN {X 0,Y 397.355,Z 273.61,A -85,B 0,C 180,E1 -11422.887,E2 -11422.887} C_VEL
LIN {X 0,Y 397.244,Z 273.624,A -85,B 0,C 180,E1 -11424.924,E2 -11424.924} C_VEL
LIN {X 0,Y 397.406,Z 273.604,A -85,B 0,C 180,E1 -11428.317,E2 -11428.317} C_VEL
LIN {X 0,Y 397.572,Z 273.585,A -85,B 0,C 180,E1 -11429.999,E2 -11429.999} C_VEL
LIN {X 0,Y 397.376,Z 273.607,A -85,B 0,C 180,E1 -11432.732,E2 -11432.732} C_VEL
LIN {X 0,Y 396.678,Z 273.701,A -85,B 0,C 180,E1 -11433.577,E2 -11433.577} C_VEL
LIN {X 0,Y 393.793,Z 274.055,A -85,B 0,C 180,E1 -11434.95,E2 -11434.95} C_VEL
LIN {X 0,Y 391.382,Z 274.355,A -85,B 0,C 180,E1 -11436.059,E2 -11436.059} C_VEL
LIN {X 0,Y 390.375,Z 274.481,A -85,B 0,C 180,E1 -11436.918,E2 -11436.918} C_VEL
LIN {X 0,Y 390.306,Z 274.491,A -85,B 0,C 180,E1 -11437.208,E2 -11437.208} C_VEL
LIN {X 0,Y 390.158,Z 274.506,A -85,B 0,C 180,E1 -11440.376,E2 -11440.376} C_VEL
LIN {X 0,Y 390.159,Z 274.512,A -85,B 0,C 180,E1 -11443.541,E2 -11443.541} C_VEL
LIN {X 0,Y 390.137,Z 274.514,A -85,B 0,C 180,E1 -11447.306,E2 -11447.306} C_VEL
LIN {X 0,Y 390.076,Z 274.516,A -85,B 0,C 180,E1 -11450.469,E2 -11450.469} C_VEL
LIN {X 0,Y 390.077,Z 274.523,A -85,B 0,C 180,E1 -11453.35,E2 -11453.35} C_VEL
LIN {X 0,Y 390.1,Z 274.514,A -85,B 0,C 180,E1 -11456.767,E2 -11456.767} C_VEL
LIN {X 0,Y 390.026,Z 274.523,A -85,B 0,C 180,E1 -11460.299,E2 -11460.299} C_VEL
LIN {X 0,Y 390.055,Z 274.52,A -85,B 0,C 180,E1 -11464.024,E2 -11464.024} C_VEL
LIN {X 0,Y 390.032,Z 274.526,A -85,B 0,C 180,E1 -11467.551,E2 -11467.551} C_VEL
LIN {X 0,Y 390.043,Z 274.522,A -85,B 0,C 180,E1 -11470.821,E2 -11470.821} C_VEL
LIN {X 0,Y 390.043,Z 274.522,A -85,B 0,C 180,E1 -11473.886,E2 -11473.886} C_VEL
LIN {X 0,Y 390.045,Z 274.522,A -85,B 0,C 180,E1 -11476.79,E2 -11476.79} C_VEL
LIN {X 0,Y 390.042,Z 274.524,A -85,B 0,C 180,E1 -11479.56,E2 -11479.56} C_VEL
LIN {X 0,Y 390.028,Z 274.523,A -85,B 0,C 180,E1 -11482.449,E2 -11482.449} C_VEL
LIN {X 0,Y 390.053,Z 274.52,A -85,B 0,C 180,E1 -11485.975,E2 -11485.975} C_VEL
LIN {X 0,Y 390.032,Z 274.523,A -85,B 0,C 180,E1 -11489.869,E2 -11489.869} C_VEL
LIN {X 0,Y 390.099,Z 274.52,A -85,B 0,C 180,E1 -11493.232,E2 -11493.232} C_VEL
LIN {X 0,Y 390.062,Z 274.521,A -85,B 0,C 180,E1 -11496.761,E2 -11496.761} C_VEL
LIN {X 0,Y 390.089,Z 274.515,A -85,B 0,C 180,E1 -11499.983,E2 -11499.983} C_VEL
LIN {X 0,Y 390.124,Z 274.516,A -85,B 0,C 180,E1 -11503.249,E2 -11503.249} C_VEL
LIN {X 0,Y 390.18,Z 274.505,A -85,B 0,C 180,E1 -11506.562,E2 -11506.562} C_VEL
LIN {X 0,Y 390.191,Z 274.505,A -85,B 0,C 180,E1 -11510.672,E2 -11510.672} C_VEL
LIN {X 0,Y 390.31,Z 274.488,A -85,B 0,C 180,E1 -11513.799,E2 -11513.799} C_VEL
LIN {X 0,Y 390.407,Z 274.475,A -85,B 0,C 180,E1 -11517.938,E2 -11517.938} C_VEL
LIN {X 0,Y 390.537,Z 274.459,A -85,B 0,C 180,E1 -11520.001,E2 -11520.001} C_VEL
LIN {X 0,Y 390.296,Z 274.495,A -85,B 0,C 180,E1 -11523.097,E2 -11523.097} C_VEL
LIN {X 0,Y 390.315,Z 274.487,A -85,B 0,C 180,E1 -11526.203,E2 -11526.203} C_VEL
LIN {X 0,Y 390.303,Z 274.489,A -85,B 0,C 180,E1 -11528.283,E2 -11528.283} C_VEL
LIN {X 0,Y 390.159,Z 274.508,A -85,B 0,C 180,E1 -11532.484,E2 -11532.484} C_VEL
LIN {X 0,Y 390.128,Z 274.51,A -85,B 0,C 180,E1 -11535.678,E2 -11535.678} C_VEL
LIN {X 0,Y 390.095,Z 274.521,A -85,B 0,C 180,E1 -11538.923,E2 -11538.923} C_VEL
LIN {X 0,Y 390.027,Z 274.523,A -85,B 0,C 180,E1 -11542.236,E2 -11542.236} C_VEL
LIN {X 0,Y 390.109,Z 274.512,A -85,B 0,C 180,E1 -11545.745,E2 -11545.745} C_VEL
LIN {X 0,Y 390.049,Z 274.524,A -85,B 0,C 180,E1 -11549.111,E2 -11549.111} C_VEL
LIN {X 0,Y 390.034,Z 274.528,A -85,B 0,C 180,E1 -11552.723,E2 -11552.723} C_VEL
LIN {X 0,Y 390.047,Z 274.52,A -85,B 0,C 180,E1 -11555.827,E2 -11555.827} C_VEL
LIN {X 0,Y 390.059,Z 274.521,A -85,B 0,C 180,E1 -11559.219,E2 -11559.219} C_VEL
LIN {X 0,Y 390.034,Z 274.524,A -85,B 0,C 180,E1 -11562.376,E2 -11562.376} C_VEL
LIN {X 0,Y 390.037,Z 274.522,A -85,B 0,C 180,E1 -11565.356,E2 -11565.356} C_VEL
LIN {X 0,Y 390.024,Z 274.524,A -85,B 0,C 180,E1 -11568.188,E2 -11568.188} C_VEL
LIN {X 0,Y 390.085,Z 274.521,A -85,B 0,C 180,E1 -11570.909,E2 -11570.909} C_VEL
LIN {X 0,Y 390.091,Z 274.712,A -85,B 0,C 180,E1 -11574.365,E2 -11574.365} C_VEL
LIN {X 0,Y 393.878,Z 289.692,A -85,B 0,C 180,E1 -11577.293,E2 -11577.293} C_VEL
LIN {X 0,Y 397.45,Z 304.434,A -85,B 0,C 180,E1 -11580.05,E2 -11580.05} C_VEL
LIN {X 0,Y 397.214,Z 309.499,A -85,B 0,C 180,E1 -11580.887,E2 -11580.887} C_VEL
LIN {X 0,Y 396.726,Z 314.409,A -85,B 0,C 180,E1 -11581.682,E2 -11581.682} C_VEL
LIN {X 0,Y 402.905,Z 352.711,A -85,B 0,C 180,E1 -11583.006,E2 -11583.006} C_VEL
LIN {X 0,Y 398.876,Z 482.032,A -85,B 0,C 180,E1 -11585.922,E2 -11585.922} C_VEL
LIN {X 0,Y 398.074,Z 497.586,A -85,B 0,C 180,E1 -11586.465,E2 -11586.465} C_VEL
LIN {X 0,Y 397.081,Z 512.005,A -85,B 0,C 180,E1 -11587.155,E2 -11587.155} C_VEL
LIN {X 0,Y 395.895,Z 527.333,A -85,B 0,C 180,E1 -11588.114,E2 -11588.114} C_VEL
LIN {X 0,Y 394.792,Z 540.538,A -85,B 0,C 180,E1 -11589.145,E2 -11589.145} C_VEL
LIN {X 0,Y 393.517,Z 554.097,A -85,B 0,C 180,E1 -11590.437,E2 -11590.437} C_VEL
LIN {X 0,Y 392.35,Z 567.007,A -85,B 0,C 180,E1 -11591.933,E2 -11591.933} C_VEL
LIN {X 0,Y 391.274,Z 578.725,A -85,B 0,C 180,E1 -11593.568,E2 -11593.568} C_VEL
LIN {X 0,Y 390.456,Z 588.194,A -85,B 0,C 180,E1 -11595.14,E2 -11595.14} C_VEL
LIN {X 0,Y 389.794,Z 596.723,A -85,B 0,C 180,E1 -11596.812,E2 -11596.812} C_VEL
LIN {X 0,Y 389.403,Z 604.12,A -85,B 0,C 180,E1 -11598.551,E2 -11598.551} C_VEL
LIN {X 0,Y 388.971,Z 611.386,A -85,B 0,C 180,E1 -11600.643,E2 -11600.643} C_VEL
LIN {X 0,Y 388.831,Z 617.029,A -85,B 0,C 180,E1 -11602.733,E2 -11602.733} C_VEL
LIN {X 0,Y 388.779,Z 621.188,A -85,B 0,C 180,E1 -11604.816,E2 -11604.816} C_VEL
LIN {X 0,Y 388.801,Z 623.963,A -85,B 0,C 180,E1 -11606.893,E2 -11606.893} C_VEL
LIN {X 0,Y 388.809,Z 625.413,A -85,B 0,C 180,E1 -11608.966,E2 -11608.966} C_VEL
LIN {X 0,Y 388.801,Z 625.573,A -85,B 0,C 180,E1 -11611.037,E2 -11611.037} C_VEL
LIN {X 0,Y 388.849,Z 625.174,A -85,B 0,C 180,E1 -11612.073,E2 -11612.073} C_VEL
LIN {X 0,Y 388.729,Z 623.398,A -85,B 0,C 180,E1 -11614.148,E2 -11614.148} C_VEL
LIN {X 0,Y 388.761,Z 620.333,A -85,B 0,C 180,E1 -11616.228,E2 -11616.228} C_VEL
LIN {X 0,Y 388.881,Z 615.905,A -85,B 0,C 180,E1 -11618.314,E2 -11618.314} C_VEL
LIN {X 0,Y 389.107,Z 610.015,A -85,B 0,C 180,E1 -11620.407,E2 -11620.407} C_VEL
LIN {X 0,Y 389.516,Z 604.525,A -85,B 0,C 180,E1 -11621.977,E2 -11621.977} C_VEL
LIN {X 0,Y 390.134,Z 596.938,A -85,B 0,C 180,E1 -11623.811,E2 -11623.811} C_VEL
LIN {X 0,Y 391.029,Z 587.83,A -85,B 0,C 180,E1 -11625.642,E2 -11625.642} C_VEL
LIN {X 0,Y 392.211,Z 576.941,A -85,B 0,C 180,E1 -11627.467,E2 -11627.467} C_VEL
LIN {X 0,Y 393.602,Z 564.841,A -85,B 0,C 180,E1 -11629.155,E2 -11629.155} C_VEL
LIN {X 0,Y 395.064,Z 552.685,A -85,B 0,C 180,E1 -11630.571,E2 -11630.571} C_VEL
LIN {X 0,Y 396.6,Z 539.632,A -85,B 0,C 180,E1 -11631.848,E2 -11631.848} C_VEL
LIN {X 0,Y 398.259,Z 524.921,A -85,B 0,C 180,E1 -11633.031,E2 -11633.031} C_VEL
LIN {X 0,Y 399.84,Z 510.392,A -85,B 0,C 180,E1 -11633.97,E2 -11633.97} C_VEL
LIN {X 0,Y 401.23,Z 495.749,A -85,B 0,C 180,E1 -11634.722,E2 -11634.722} C_VEL
LIN {X 0,Y 402.624,Z 479.087,A -85,B 0,C 180,E1 -11635.355,E2 -11635.355} C_VEL
LIN {X 0,Y 407.931,Z 384.446,A -85,B 0,C 180,E1 -11637.899,E2 -11637.899} C_VEL
LIN {X 0,Y 409.866,Z 353.534,A -85,B 0,C 180,E1 -11638.782,E2 -11638.782} C_VEL
LIN {X 0,Y 408.33,Z 338.868,A -85,B 0,C 180,E1 -11639.527,E2 -11639.527} C_VEL
LIN {X 0,Y 405.889,Z 323.379,A -85,B 0,C 180,E1 -11640.484,E2 -11640.484} C_VEL
LIN {X 0,Y 403.995,Z 314.353,A -85,B 0,C 180,E1 -11641.147,E2 -11641.147} C_VEL
LIN {X 0,Y 401.878,Z 309.639,A -85,B 0,C 180,E1 -11641.694,E2 -11641.694} C_VEL
LIN {X 0,Y 399.618,Z 304.761,A -85,B 0,C 180,E1 -11642.336,E2 -11642.336} C_VEL
LIN {X 0,Y 397.898,Z 297.434,A -85,B 0,C 180,E1 -11644.418,E2 -11644.418} C_VEL
LIN {X 0,Y 396.017,Z 291.264,A -85,B 0,C 180,E1 -11646.509,E2 -11646.509} C_VEL
LIN {X 0,Y 394.384,Z 286.176,A -85,B 0,C 180,E1 -11648.589,E2 -11648.589} C_VEL
LIN {X 0,Y 393.029,Z 282.495,A -85,B 0,C 180,E1 -11650.496,E2 -11650.496} C_VEL
LIN {X 0,Y 392.445,Z 280.884,A -85,B 0,C 180,E1 -11651.5,E2 -11651.5} C_VEL
LIN {X 0,Y 391.157,Z 277.51,A -85,B 0,C 180,E1 -11654.486,E2 -11654.486} C_VEL
LIN {X 0,Y 390.561,Z 276.394,A -85,B 0,C 180,E1 -11656.858,E2 -11656.858} C_VEL
LIN {X 0,Y 390.649,Z 276.537,A -85,B 0,C 180,E1 -11659.634,E2 -11659.634} C_VEL
LIN {X 0,Y 391.371,Z 278.069,A -85,B 0,C 180,E1 -11662.199,E2 -11662.199} C_VEL
LIN {X 0,Y 392.568,Z 281.476,A -85,B 0,C 180,E1 -11665.048,E2 -11665.048} C_VEL
LIN {X 0,Y 393.534,Z 284.265,A -85,B 0,C 180,E1 -11666.643,E2 -11666.643} C_VEL
LIN {X 0,Y 397.469,Z 289.553,A -85,B 0,C 180,E1 -11667.76,E2 -11667.76} C_VEL
LIN {X 0,Y 400.634,Z 294.042,A -85,B 0,C 180,E1 -11668.571,E2 -11668.571} C_VEL
LIN {X 0,Y 404.775,Z 300.357,A -85,B 0,C 180,E1 -11669.559,E2 -11669.559} C_VEL
LIN {X 0,Y 409.944,Z 309.61,A -85,B 0,C 180,E1 -11670.722,E2 -11670.722} C_VEL
LIN {X 0,Y 411.837,Z 313.573,A -85,B 0,C 180,E1 -11671.133,E2 -11671.133} C_VEL
LIN {X 0,Y 406.387,Z 392.072,A -85,B 0,C 180,E1 -11673.348,E2 -11673.348} C_VEL
LIN {X 0,Y 403.614,Z 443.863,A -85,B 0,C 180,E1 -11674.764,E2 -11674.764} C_VEL
LIN {X 0,Y 402.578,Z 458.959,A -85,B 0,C 180,E1 -11675.36,E2 -11675.36} C_VEL
LIN {X 0,Y 401.39,Z 473.998,A -85,B 0,C 180,E1 -11676.16,E2 -11676.16} C_VEL
LIN {X 0,Y 400.144,Z 488.201,A -85,B 0,C 180,E1 -11677.132,E2 -11677.132} C_VEL
LIN {X 0,Y 398.712,Z 501.827,A -85,B 0,C 180,E1 -11678.274,E2 -11678.274} C_VEL
LIN {X 0,Y 397.099,Z 515.407,A -85,B 0,C 180,E1 -11679.661,E2 -11679.661} C_VEL
LIN {X 0,Y 395.538,Z 526.935,A -85,B 0,C 180,E1 -11681.078,E2 -11681.078} C_VEL
LIN {X 0,Y 394.272,Z 537.424,A -85,B 0,C 180,E1 -11682.627,E2 -11682.627} C_VEL
LIN {X 0,Y 392.912,Z 547.672,A -85,B 0,C 180,E1 -11684.436,E2 -11684.436} C_VEL
LIN {X 0,Y 391.705,Z 556.172,A -85,B 0,C 180,E1 -11686.247,E2 -11686.247} C_VEL
LIN {X 0,Y 390.911,Z 563.187,A -85,B 0,C 180,E1 -11688.067,E2 -11688.067} C_VEL
LIN {X 0,Y 390.143,Z 569.646,A -85,B 0,C 180,E1 -11690.146,E2 -11690.146} C_VEL
LIN {X 0,Y 389.62,Z 574.618,A -85,B 0,C 180,E1 -11692.224,E2 -11692.224} C_VEL
LIN {X 0,Y 389.297,Z 577.458,A -85,B 0,C 180,E1 -11693.781,E2 -11693.781} C_VEL
LIN {X 0,Y 389.153,Z 580.073,A -85,B 0,C 180,E1 -11695.857,E2 -11695.857} C_VEL
LIN {X 0,Y 388.942,Z 581.46,A -85,B 0,C 180,E1 -11697.928,E2 -11697.928} C_VEL
LIN {X 0,Y 388.803,Z 581.619,A -85,B 0,C 180,E1 -11699.999,E2 -11699.999} C_VEL
LIN {X 0,Y 388.9,Z 580.544,A -85,B 0,C 180,E1 -11702.07,E2 -11702.07} C_VEL
LIN {X 0,Y 388.907,Z 578.237,A -85,B 0,C 180,E1 -11704.144,E2 -11704.144} C_VEL
LIN {X 0,Y 389.099,Z 574.631,A -85,B 0,C 180,E1 -11706.221,E2 -11706.221} C_VEL
LIN {X 0,Y 389.336,Z 569.648,A -85,B 0,C 180,E1 -11708.302,E2 -11708.302} C_VEL
LIN {X 0,Y 389.751,Z 563.156,A -85,B 0,C 180,E1 -11710.387,E2 -11710.387} C_VEL
LIN {X 0,Y 390.371,Z 556.102,A -85,B 0,C 180,E1 -11712.212,E2 -11712.212} C_VEL
LIN {X 0,Y 391.076,Z 547.088,A -85,B 0,C 180,E1 -11714.131,E2 -11714.131} C_VEL
LIN {X 0,Y 391.952,Z 537.236,A -85,B 0,C 180,E1 -11715.868,E2 -11715.868} C_VEL
LIN {X 0,Y 392.917,Z 526.649,A -85,B 0,C 180,E1 -11717.433,E2 -11717.433} C_VEL
LIN {X 0,Y 393.992,Z 515.118,A -85,B 0,C 180,E1 -11718.865,E2 -11718.865} C_VEL
LIN {X 0,Y 395.042,Z 502.685,A -85,B 0,C 180,E1 -11720.162,E2 -11720.162} C_VEL
LIN {X 0,Y 396.156,Z 489.209,A -85,B 0,C 180,E1 -11721.325,E2 -11721.325} C_VEL
LIN {X 0,Y 397.21,Z 474.449,A -85,B 0,C 180,E1 -11722.358,E2 -11722.358} C_VEL
LIN {X 0,Y 398.17,Z 458.633,A -85,B 0,C 180,E1 -11723.216,E2 -11723.216} C_VEL
LIN {X 0,Y 398.847,Z 443.111,A -85,B 0,C 180,E1 -11723.84,E2 -11723.84} C_VEL
LIN {X 0,Y 399.396,Z 426.565,A -85,B 0,C 180,E1 -11724.287,E2 -11724.287} C_VEL
LIN {X 0,Y 403.114,Z 305.686,A -85,B 0,C 180,E1 -11726.985,E2 -11726.985} C_VEL
LIN {X 0,Y 395.974,Z 288.247,A -85,B 0,C 180,E1 -11727.851,E2 -11727.851} C_VEL
LIN {X 0,Y 390.142,Z 275.051,A -85,B 0,C 180,E1 -11728.557,E2 -11728.557} C_VEL
LIN {X 0,Y 390.039,Z 274.525,A -85,B 0,C 180,E1 -11728.593,E2 -11728.593} C_VEL
LIN {X 0,Y 390.033,Z 274.527,A -85,B 0,C 180,E1 -11732.123,E2 -11732.123} C_VEL
LIN {X 0,Y 390.085,Z 274.516,A -85,B 0,C 180,E1 -11735.206,E2 -11735.206} C_VEL
LIN {X 0,Y 390.062,Z 274.519,A -85,B 0,C 180,E1 -11739.094,E2 -11739.094} C_VEL
LIN {X 0,Y 390.037,Z 274.523,A -85,B 0,C 180,E1 -11742.372,E2 -11742.372} C_VEL
LIN {X 0,Y 390.042,Z 274.523,A -85,B 0,C 180,E1 -11745.353,E2 -11745.353} C_VEL
LIN {X 0,Y 390.029,Z 274.525,A -85,B 0,C 180,E1 -11748.185,E2 -11748.185} C_VEL
LIN {X 0,Y 390.085,Z 274.515,A -85,B 0,C 180,E1 -11750.906,E2 -11750.906} C_VEL
LIN {X 0,Y 390.081,Z 274.516,A -85,B 0,C 180,E1 -11754.791,E2 -11754.791} C_VEL
LIN {X 0,Y 390.019,Z 274.524,A -85,B 0,C 180,E1 -11758.494,E2 -11758.494} C_VEL
LIN {X 0,Y 390.035,Z 274.525,A -85,B 0,C 180,E1 -11762.062,E2 -11762.062} C_VEL
LIN {X 0,Y 390.056,Z 274.524,A -85,B 0,C 180,E1 -11765.516,E2 -11765.516} C_VEL
LIN {X 0,Y 390.05,Z 274.52,A -85,B 0,C 180,E1 -11768.876,E2 -11768.876} C_VEL
LIN {X 0,Y 390.106,Z 274.515,A -85,B 0,C 180,E1 -11772.164,E2 -11772.164} C_VEL
LIN {X 0,Y 390.138,Z 274.513,A -85,B 0,C 180,E1 -11775.391,E2 -11775.391} C_VEL
LIN {X 0,Y 390.141,Z 274.508,A -85,B 0,C 180,E1 -11778.57,E2 -11778.57} C_VEL
LIN {X 0,Y 390.337,Z 274.487,A -85,B 0,C 180,E1 -11781.992,E2 -11781.992} C_VEL
LIN {X 0,Y 390.216,Z 274.499,A -85,B 0,C 180,E1 -11784.832,E2 -11784.832} C_VEL
LIN {X 0,Y 390.409,Z 274.478,A -85,B 0,C 180,E1 -11787.935,E2 -11787.935} C_VEL
LIN {X 0,Y 390.541,Z 274.461,A -85,B 0,C 180,E1 -11789.999,E2 -11789.999} C_VEL
LIN {X 0,Y 390.301,Z 274.491,A -85,B 0,C 180,E1 -11793.095,E2 -11793.095} C_VEL
LIN {X 0,Y 390.306,Z 274.491,A -85,B 0,C 180,E1 -11797.208,E2 -11797.208} C_VEL
LIN {X 0,Y 389.656,Z 274.58,A -85,B 0,C 180,E1 -11798.068,E2 -11798.068} C_VEL
LIN {X 0,Y 386.739,Z 274.949,A -85,B 0,C 180,E1 -11799.465,E2 -11799.465} C_VEL
LIN {X 0,Y 384.246,Z 275.256,A -85,B 0,C 180,E1 -11800.593,E2 -11800.593} C_VEL
LIN {X 0,Y 383.173,Z 275.383,A -85,B 0,C 180,E1 -11801.467,E2 -11801.467} C_VEL
LIN {X 0,Y 383.085,Z 275.391,A -85,B 0,C 180,E1 -11801.764,E2 -11801.764} C_VEL
LIN {X 0,Y 383.099,Z 275.387,A -85,B 0,C 180,E1 -11804.88,E2 -11804.88} C_VEL
LIN {X 0,Y 383.051,Z 275.392,A -85,B 0,C 180,E1 -11808.172,E2 -11808.172} C_VEL
LIN {X 0,Y 382.987,Z 275.405,A -85,B 0,C 180,E1 -11811.53,E2 -11811.53} C_VEL
LIN {X 0,Y 383.039,Z 275.395,A -85,B 0,C 180,E1 -11814.959,E2 -11814.959} C_VEL
LIN {X 0,Y 383.017,Z 275.396,A -85,B 0,C 180,E1 -11818.269,E2 -11818.269} C_VEL
LIN {X 0,Y 382.996,Z 275.399,A -85,B 0,C 180,E1 -11822.149,E2 -11822.149} C_VEL
LIN {X 0,Y 383.005,Z 275.398,A -85,B 0,C 180,E1 -11824.667,E2 -11824.667} C_VEL
LIN {X 0,Y 382.988,Z 275.401,A -85,B 0,C 180,E1 -11827.903,E2 -11827.903} C_VEL
LIN {X 0,Y 382.971,Z 275.408,A -85,B 0,C 180,E1 -11831.347,E2 -11831.347} C_VEL
LIN {X 0,Y 382.985,Z 275.4,A -85,B 0,C 180,E1 -11834.303,E2 -11834.303} C_VEL
LIN {X 0,Y 382.996,Z 275.405,A -85,B 0,C 180,E1 -11837.24,E2 -11837.24} C_VEL
LIN {X 0,Y 383,Z 275.398,A -85,B 0,C 180,E1 -11840.413,E2 -11840.413} C_VEL
LIN {X 0,Y 383.01,Z 275.397,A -85,B 0,C 180,E1 -11844.044,E2 -11844.044} C_VEL
LIN {X 0,Y 382.972,Z 275.404,A -85,B 0,C 180,E1 -11847.578,E2 -11847.578} C_VEL
LIN {X 0,Y 382.977,Z 275.401,A -85,B 0,C 180,E1 -11850.3,E2 -11850.3} C_VEL
LIN {X 0,Y 383.066,Z 275.39,A -85,B 0,C 180,E1 -11854.021,E2 -11854.021} C_VEL
LIN {X 0,Y 382.981,Z 275.405,A -85,B 0,C 180,E1 -11857.335,E2 -11857.335} C_VEL
LIN {X 0,Y 383.046,Z 275.395,A -85,B 0,C 180,E1 -11860.717,E2 -11860.717} C_VEL
LIN {X 0,Y 383.066,Z 275.39,A -85,B 0,C 180,E1 -11864.027,E2 -11864.027} C_VEL
LIN {X 0,Y 383.122,Z 275.387,A -85,B 0,C 180,E1 -11867.284,E2 -11867.284} C_VEL
LIN {X 0,Y 383.138,Z 275.382,A -85,B 0,C 180,E1 -11870.498,E2 -11870.498} C_VEL
LIN {X 0,Y 383.266,Z 275.366,A -85,B 0,C 180,E1 -11873.684,E2 -11873.684} C_VEL
LIN {X 0,Y 383.375,Z 275.351,A -85,B 0,C 180,E1 -11877.9,E2 -11877.9} C_VEL
LIN {X 0,Y 383.506,Z 275.335,A -85,B 0,C 180,E1 -11880.001,E2 -11880.001} C_VEL
LIN {X 0,Y 383.233,Z 275.374,A -85,B 0,C 180,E1 -11883.155,E2 -11883.155} C_VEL
LIN {X 0,Y 383.272,Z 275.365,A -85,B 0,C 180,E1 -11886.317,E2 -11886.317} C_VEL
LIN {X 0,Y 383.248,Z 275.369,A -85,B 0,C 180,E1 -11888.437,E2 -11888.437} C_VEL
LIN {X 0,Y 383.086,Z 275.388,A -85,B 0,C 180,E1 -11891.643,E2 -11891.643} C_VEL
LIN {X 0,Y 383.098,Z 275.392,A -85,B 0,C 180,E1 -11894.883,E2 -11894.883} C_VEL
LIN {X 0,Y 383.052,Z 275.392,A -85,B 0,C 180,E1 -11898.175,E2 -11898.175} C_VEL
LIN {X 0,Y 382.981,Z 275.401,A -85,B 0,C 180,E1 -11901.532,E2 -11901.532} C_VEL
LIN {X 0,Y 383.041,Z 275.399,A -85,B 0,C 180,E1 -11904.962,E2 -11904.962} C_VEL
LIN {X 0,Y 383.031,Z 275.397,A -85,B 0,C 180,E1 -11908.494,E2 -11908.494} C_VEL
LIN {X 0,Y 383,Z 275.399,A -85,B 0,C 180,E1 -11912.151,E2 -11912.151} C_VEL
LIN {X 0,Y 383.009,Z 275.402,A -85,B 0,C 180,E1 -11914.669,E2 -11914.669} C_VEL
LIN {X 0,Y 382.99,Z 275.399,A -85,B 0,C 180,E1 -11917.905,E2 -11917.905} C_VEL
LIN {X 0,Y 382.976,Z 275.402,A -85,B 0,C 180,E1 -11921.349,E2 -11921.349} C_VEL
LIN {X 0,Y 382.988,Z 275.402,A -85,B 0,C 180,E1 -11924.305,E2 -11924.305} C_VEL
LIN {X 0,Y 383.004,Z 275.399,A -85,B 0,C 180,E1 -11927.242,E2 -11927.242} C_VEL
LIN {X 0,Y 383.009,Z 275.403,A -85,B 0,C 180,E1 -11930.415,E2 -11930.415} C_VEL
LIN {X 0,Y 383.019,Z 275.499,A -85,B 0,C 180,E1 -11933.961,E2 -11933.961} C_VEL
LIN {X 0,Y 386.859,Z 290.611,A -85,B 0,C 180,E1 -11936.977,E2 -11936.977} C_VEL
LIN {X 0,Y 390.625,Z 306.418,A -85,B 0,C 180,E1 -11939.98,E2 -11939.98} C_VEL
LIN {X 0,Y 389.948,Z 314.079,A -85,B 0,C 180,E1 -11941.249,E2 -11941.249} C_VEL
LIN {X 0,Y 396.254,Z 353.902,A -85,B 0,C 180,E1 -11942.655,E2 -11942.655} C_VEL
LIN {X 0,Y 392.11,Z 481.813,A -85,B 0,C 180,E1 -11945.621,E2 -11945.621} C_VEL
LIN {X 0,Y 391.245,Z 497.453,A -85,B 0,C 180,E1 -11946.18,E2 -11946.18} C_VEL
LIN {X 0,Y 390.18,Z 512.734,A -85,B 0,C 180,E1 -11946.937,E2 -11946.937} C_VEL
LIN {X 0,Y 389.03,Z 526.935,A -85,B 0,C 180,E1 -11947.847,E2 -11947.847} C_VEL
LIN {X 0,Y 387.894,Z 540.141,A -85,B 0,C 180,E1 -11948.895,E2 -11948.895} C_VEL
LIN {X 0,Y 386.586,Z 553.707,A -85,B 0,C 180,E1 -11950.21,E2 -11950.21} C_VEL
LIN {X 0,Y 385.449,Z 565.439,A -85,B 0,C 180,E1 -11951.575,E2 -11951.575} C_VEL
LIN {X 0,Y 384.348,Z 577.511,A -85,B 0,C 180,E1 -11953.264,E2 -11953.264} C_VEL
LIN {X 0,Y 383.475,Z 587.125,A -85,B 0,C 180,E1 -11954.863,E2 -11954.863} C_VEL
LIN {X 0,Y 382.745,Z 596.389,A -85,B 0,C 180,E1 -11956.704,E2 -11956.704} C_VEL
LIN {X 0,Y 382.297,Z 604.294,A -85,B 0,C 180,E1 -11958.604,E2 -11958.604} C_VEL
LIN {X 0,Y 381.915,Z 610.614,A -85,B 0,C 180,E1 -11960.468,E2 -11960.468} C_VEL
LIN {X 0,Y 381.774,Z 616.349,A -85,B 0,C 180,E1 -11962.598,E2 -11962.598} C_VEL
LIN {X 0,Y 381.702,Z 620.585,A -85,B 0,C 180,E1 -11964.719,E2 -11964.719} C_VEL
LIN {X 0,Y 381.707,Z 623.428,A -85,B 0,C 180,E1 -11966.835,E2 -11966.835} C_VEL
LIN {X 0,Y 381.782,Z 624.353,A -85,B 0,C 180,E1 -11967.892,E2 -11967.892} C_VEL
LIN {X 0,Y 381.725,Z 625.21,A -85,B 0,C 180,E1 -11970.001,E2 -11970.001} C_VEL
LIN {X 0,Y 381.779,Z 624.781,A -85,B 0,C 180,E1 -11972.111,E2 -11972.111} C_VEL
LIN {X 0,Y 381.651,Z 623.053,A -85,B 0,C 180,E1 -11974.226,E2 -11974.226} C_VEL
LIN {X 0,Y 381.667,Z 620.025,A -85,B 0,C 180,E1 -11976.345,E2 -11976.345} C_VEL
LIN {X 0,Y 381.79,Z 615.629,A -85,B 0,C 180,E1 -11978.47,E2 -11978.47} C_VEL
LIN {X 0,Y 382.064,Z 609.78,A -85,B 0,C 180,E1 -11980.601,E2 -11980.601} C_VEL
LIN {X 0,Y 382.663,Z 602.365,A -85,B 0,C 180,E1 -11982.733,E2 -11982.733} C_VEL
LIN {X 0,Y 383.39,Z 594.413,A -85,B 0,C 180,E1 -11984.6,E2 -11984.6} C_VEL
LIN {X 0,Y 384.458,Z 584.91,A -85,B 0,C 180,E1 -11986.461,E2 -11986.461} C_VEL
LIN {X 0,Y 385.726,Z 574.121,A -85,B 0,C 180,E1 -11988.231,E2 -11988.231} C_VEL
LIN {X 0,Y 387.264,Z 561.989,A -85,B 0,C 180,E1 -11989.895,E2 -11989.895} C_VEL
LIN {X 0,Y 389.005,Z 548.239,A -85,B 0,C 180,E1 -11991.461,E2 -11991.461} C_VEL
LIN {X 0,Y 390.789,Z 534.442,A -85,B 0,C 180,E1 -11992.748,E2 -11992.748} C_VEL
LIN {X 0,Y 392.469,Z 520.094,A -85,B 0,C 180,E1 -11993.853,E2 -11993.853} C_VEL
LIN {X 0,Y 394.288,Z 503.902,A -85,B 0,C 180,E1 -11994.835,E2 -11994.835} C_VEL
LIN {X 0,Y 395.817,Z 488.751,A -85,B 0,C 180,E1 -11995.541,E2 -11995.541} C_VEL
LIN {X 0,Y 397.143,Z 470.764,A -85,B 0,C 180,E1 -11996.153,E2 -11996.153} C_VEL
LIN {X 0,Y 401.747,Z 394.013,A -85,B 0,C 180,E1 -11998.262,E2 -11998.262} C_VEL
LIN {X 0,Y 404.49,Z 355.079,A -85,B 0,C 180,E1 -11999.395,E2 -11999.395} C_VEL
LIN {X 0,Y 403.122,Z 340.86,A -85,B 0,C 180,E1 -12000.148,E2 -12000.148} C_VEL
LIN {X 0,Y 400.77,Z 325.002,A -85,B 0,C 180,E1 -12001.177,E2 -12001.177} C_VEL
LIN {X 0,Y 399.366,Z 318.11,A -85,B 0,C 180,E1 -12001.714,E2 -12001.714} C_VEL
LIN {X 0,Y 397.404,Z 313.762,A -85,B 0,C 180,E1 -12002.254,E2 -12002.254} C_VEL
LIN {X 0,Y 394.882,Z 308.607,A -85,B 0,C 180,E1 -12002.967,E2 -12002.967} C_VEL
LIN {X 0,Y 392.477,Z 303.632,A -85,B 0,C 180,E1 -12003.72,E2 -12003.72} C_VEL
LIN {X 0,Y 390.625,Z 296.806,A -85,B 0,C 180,E1 -12005.94,E2 -12005.94} C_VEL
LIN {X 0,Y 388.689,Z 290.597,A -85,B 0,C 180,E1 -12008.45,E2 -12008.45} C_VEL
LIN {X 0,Y 387.127,Z 286.148,A -85,B 0,C 180,E1 -12010.811,E2 -12010.811} C_VEL
LIN {X 0,Y 385.881,Z 282.962,A -85,B 0,C 180,E1 -12013.237,E2 -12013.237} C_VEL
LIN {X 0,Y 385.164,Z 281.273,A -85,B 0,C 180,E1 -12015.369,E2 -12015.369} C_VEL
LIN {X 0,Y 384.83,Z 280.572,A -85,B 0,C 180,E1 -12017.49,E2 -12017.49} C_VEL
LIN {X 0,Y 385.08,Z 281.024,A -85,B 0,C 180,E1 -12020.299,E2 -12020.299} C_VEL
LIN {X 0,Y 385.434,Z 281.849,A -85,B 0,C 180,E1 -12021.686,E2 -12021.686} C_VEL
LIN {X 0,Y 386.386,Z 284.669,A -85,B 0,C 180,E1 -12024.405,E2 -12024.405} C_VEL
LIN {X 0,Y 386.863,Z 285.775,A -85,B 0,C 180,E1 -12025.116,E2 -12025.116} C_VEL
LIN {X 0,Y 389.927,Z 289.695,A -85,B 0,C 180,E1 -12026.157,E2 -12026.157} C_VEL
LIN {X 0,Y 394.145,Z 295.395,A -85,B 0,C 180,E1 -12027.415,E2 -12027.415} C_VEL
LIN {X 0,Y 397.383,Z 300.116,A -85,B 0,C 180,E1 -12028.29,E2 -12028.29} C_VEL
LIN {X 0,Y 401.822,Z 307.289,A -85,B 0,C 180,E1 -12029.403,E2 -12029.403} C_VEL
LIN {X 0,Y 406.43,Z 316.061,A -85,B 0,C 180,E1 -12030.492,E2 -12030.492} C_VEL
LIN {X 0,Y 404.746,Z 338.337,A -85,B 0,C 180,E1 -12031.171,E2 -12031.171} C_VEL
LIN {X 0,Y 399.6,Z 410.792,A -85,B 0,C 180,E1 -12033.247,E2 -12033.247} C_VEL
LIN {X 0,Y 397.671,Z 445.268,A -85,B 0,C 180,E1 -12034.237,E2 -12034.237} C_VEL
LIN {X 0,Y 396.502,Z 460.84,A -85,B 0,C 180,E1 -12034.882,E2 -12034.882} C_VEL
LIN {X 0,Y 395.16,Z 476.331,A -85,B 0,C 180,E1 -12035.747,E2 -12035.747} C_VEL
LIN {X 0,Y 393.818,Z 490.253,A -85,B 0,C 180,E1 -12036.743,E2 -12036.743} C_VEL
LIN {X 0,Y 392.312,Z 503.545,A -85,B 0,C 180,E1 -12037.901,E2 -12037.901} C_VEL
LIN {X 0,Y 390.793,Z 515.433,A -85,B 0,C 180,E1 -12039.143,E2 -12039.143} C_VEL
LIN {X 0,Y 389.267,Z 526.306,A -85,B 0,C 180,E1 -12040.487,E2 -12040.487} C_VEL
LIN {X 0,Y 387.794,Z 536.965,A -85,B 0,C 180,E1 -12042.055,E2 -12042.055} C_VEL
LIN {X 0,Y 386.376,Z 547.34,A -85,B 0,C 180,E1 -12043.895,E2 -12043.895} C_VEL
LIN {X 0,Y 385.032,Z 555.976,A -85,B 0,C 180,E1 -12045.734,E2 -12045.734} C_VEL
LIN {X 0,Y 384.002,Z 564.01,A -85,B 0,C 180,E1 -12047.849,E2 -12047.849} C_VEL
LIN {X 0,Y 383.168,Z 570.391,A -85,B 0,C 180,E1 -12049.964,E2 -12049.964} C_VEL
LIN {X 0,Y 382.606,Z 575.285,A -85,B 0,C 180,E1 -12052.081,E2 -12052.081} C_VEL
LIN {X 0,Y 382.268,Z 578.086,A -85,B 0,C 180,E1 -12053.666,E2 -12053.666} C_VEL
LIN {X 0,Y 382.082,Z 580.634,A -85,B 0,C 180,E1 -12055.78,E2 -12055.78} C_VEL
LIN {X 0,Y 381.877,Z 581.948,A -85,B 0,C 180,E1 -12057.89,E2 -12057.89} C_VEL
LIN {X 0,Y 381.73,Z 582.035,A -85,B 0,C 180,E1 -12059.999,E2 -12059.999} C_VEL
LIN {X 0,Y 381.835,Z 580.883,A -85,B 0,C 180,E1 -12062.109,E2 -12062.109} C_VEL
LIN {X 0,Y 381.827,Z 578.493,A -85,B 0,C 180,E1 -12064.221,E2 -12064.221} C_VEL
LIN {X 0,Y 382.028,Z 574.799,A -85,B 0,C 180,E1 -12066.336,E2 -12066.336} C_VEL
LIN {X 0,Y 382.279,Z 569.719,A -85,B 0,C 180,E1 -12068.457,E2 -12068.457} C_VEL
LIN {X 0,Y 382.722,Z 563.117,A -85,B 0,C 180,E1 -12070.58,E2 -12070.58} C_VEL
LIN {X 0,Y 383.381,Z 555.966,A -85,B 0,C 180,E1 -12072.438,E2 -12072.438} C_VEL
LIN {X 0,Y 384.083,Z 547.165,A -85,B 0,C 180,E1 -12074.324,E2 -12074.324} C_VEL
LIN {X 0,Y 385.046,Z 536.792,A -85,B 0,C 180,E1 -12076.161,E2 -12076.161} C_VEL
LIN {X 0,Y 386.065,Z 526.049,A -85,B 0,C 180,E1 -12077.752,E2 -12077.752} C_VEL
LIN {X 0,Y 387.058,Z 515.495,A -85,B 0,C 180,E1 -12079.076,E2 -12079.076} C_VEL
LIN {X 0,Y 388.156,Z 503.029,A -85,B 0,C 180,E1 -12080.397,E2 -12080.397} C_VEL
LIN {X 0,Y 389.304,Z 489.544,A -85,B 0,C 180,E1 -12081.58,E2 -12081.58} C_VEL
LIN {X 0,Y 390.378,Z 474.78,A -85,B 0,C 180,E1 -12082.631,E2 -12082.631} C_VEL
LIN {X 0,Y 391.37,Z 459.114,A -85,B 0,C 180,E1 -12083.497,E2 -12083.497} C_VEL
LIN {X 0,Y 392.083,Z 443.309,A -85,B 0,C 180,E1 -12084.143,E2 -12084.143} C_VEL
LIN {X 0,Y 392.646,Z 427.099,A -85,B 0,C 180,E1 -12084.591,E2 -12084.591} C_VEL
LIN {X 0,Y 396.565,Z 308.068,A -85,B 0,C 180,E1 -12087.31,E2 -12087.31} C_VEL
LIN {X 0,Y 393.953,Z 300.9,A -85,B 0,C 180,E1 -12087.65,E2 -12087.65} C_VEL
LIN {X 0,Y 385.154,Z 280.878,A -85,B 0,C 180,E1 -12088.719,E2 -12088.719} C_VEL
LIN {X 0,Y 383.164,Z 276.232,A -85,B 0,C 180,E1 -12088.973,E2 -12088.973} C_VEL
LIN {X 0,Y 383.008,Z 275.4,A -85,B 0,C 180,E1 -12089.043,E2 -12089.043} C_VEL
LIN {X 0,Y 382.988,Z 275.404,A -85,B 0,C 180,E1 -12092.42,E2 -12092.42} C_VEL
LIN {X 0,Y 383.025,Z 275.401,A -85,B 0,C 180,E1 -12095.954,E2 -12095.954} C_VEL
LIN {X 0,Y 382.992,Z 275.403,A -85,B 0,C 180,E1 -12099.581,E2 -12099.581} C_VEL
LIN {X 0,Y 383.005,Z 275.397,A -85,B 0,C 180,E1 -12102.777,E2 -12102.777} C_VEL
LIN {X 0,Y 382.996,Z 275.405,A -85,B 0,C 180,E1 -12105.788,E2 -12105.788} C_VEL
LIN {X 0,Y 382.986,Z 275.4,A -85,B 0,C 180,E1 -12108.794,E2 -12108.794} C_VEL
LIN {X 0,Y 382.996,Z 275.402,A -85,B 0,C 180,E1 -12112.095,E2 -12112.095} C_VEL
LIN {X 0,Y 383.015,Z 275.398,A -85,B 0,C 180,E1 -12115.33,E2 -12115.33} C_VEL
LIN {X 0,Y 382.978,Z 275.401,A -85,B 0,C 180,E1 -12119.08,E2 -12119.08} C_VEL
LIN {X 0,Y 382.989,Z 275.399,A -85,B 0,C 180,E1 -12122.692,E2 -12122.692} C_VEL
LIN {X 0,Y 383.012,Z 275.398,A -85,B 0,C 180,E1 -12126.19,E2 -12126.19} C_VEL
LIN {X 0,Y 383.05,Z 275.398,A -85,B 0,C 180,E1 -12129.597,E2 -12129.597} C_VEL
LIN {X 0,Y 383.088,Z 275.387,A -85,B 0,C 180,E1 -12132.929,E2 -12132.929} C_VEL
LIN {X 0,Y 383.119,Z 275.383,A -85,B 0,C 180,E1 -12136.462,E2 -12136.462} C_VEL
LIN {X 0,Y 383.145,Z 275.38,A -85,B 0,C 180,E1 -12140.496,E2 -12140.496} C_VEL
LIN {X 0,Y 383.265,Z 275.365,A -85,B 0,C 180,E1 -12142.624,E2 -12142.624} C_VEL
LIN {X 0,Y 383.188,Z 275.375,A -85,B 0,C 180,E1 -12144.737,E2 -12144.737} C_VEL
LIN {X 0,Y 383.376,Z 275.354,A -85,B 0,C 180,E1 -12147.897,E2 -12147.897} C_VEL
LIN {X 0,Y 383.511,Z 275.337,A -85,B 0,C 180,E1 -12149.999,E2 -12149.999} C_VEL
LIN {X 0,Y 383.237,Z 275.371,A -85,B 0,C 180,E1 -12153.152,E2 -12153.152} C_VEL
LIN {X 0,Y 383.256,Z 275.37,A -85,B 0,C 180,E1 -12157.213,E2 -12157.213} C_VEL
LIN {X 0,Y 383.121,Z 275.383,A -85,B 0,C 180,E1 -12160.569,E2 -12160.569} C_VEL
LIN {X 0,Y 383.085,Z 275.391,A -85,B 0,C 180,E1 -12161.764,E2 -12161.764} C_VEL
LIN {X 0,Y 382.418,Z 275.472,A -85,B 0,C 180,E1 -12162.641,E2 -12162.641} C_VEL
LIN {X 0,Y 379.567,Z 275.827,A -85,B 0,C 180,E1 -12164.067,E2 -12164.067} C_VEL
LIN {X 0,Y 377.148,Z 276.131,A -85,B 0,C 180,E1 -12165.22,E2 -12165.22} C_VEL
LIN {X 0,Y 376.102,Z 276.258,A -85,B 0,C 180,E1 -12166.111,E2 -12166.111} C_VEL
LIN {X 0,Y 376.013,Z 276.268,A -85,B 0,C 180,E1 -12166.413,E2 -12166.413} C_VEL
LIN {X 0,Y 375.987,Z 276.276,A -85,B 0,C 180,E1 -12169.659,E2 -12169.659} C_VEL
LIN {X 0,Y 375.983,Z 276.276,A -85,B 0,C 180,E1 -12173.666,E2 -12173.666} C_VEL
LIN {X 0,Y 376.007,Z 276.27,A -85,B 0,C 180,E1 -12176.651,E2 -12176.651} C_VEL
LIN {X 0,Y 375.952,Z 276.276,A -85,B 0,C 180,E1 -12180.312,E2 -12180.312} C_VEL
LIN {X 0,Y 375.946,Z 276.277,A -85,B 0,C 180,E1 -12184.111,E2 -12184.111} C_VEL
LIN {X 0,Y 375.941,Z 276.278,A -85,B 0,C 180,E1 -12186.74,E2 -12186.74} C_VEL
LIN {X 0,Y 375.975,Z 276.274,A -85,B 0,C 180,E1 -12189.97,E2 -12189.97} C_VEL
LIN {X 0,Y 375.918,Z 276.282,A -85,B 0,C 180,E1 -12193.765,E2 -12193.765} C_VEL
LIN {X 0,Y 375.92,Z 276.282,A -85,B 0,C 180,E1 -12196.81,E2 -12196.81} C_VEL
LIN {X 0,Y 375.947,Z 276.277,A -85,B 0,C 180,E1 -12200.537,E2 -12200.537} C_VEL
LIN {X 0,Y 375.949,Z 276.28,A -85,B 0,C 180,E1 -12203.495,E2 -12203.495} C_VEL
LIN {X 0,Y 375.945,Z 276.278,A -85,B 0,C 180,E1 -12205.888,E2 -12205.888} C_VEL
LIN {X 0,Y 375.95,Z 276.278,A -85,B 0,C 180,E1 -12209.687,E2 -12209.687} C_VEL
LIN {X 0,Y 376.005,Z 276.274,A -85,B 0,C 180,E1 -12213.348,E2 -12213.348} C_VEL
LIN {X 0,Y 375.969,Z 276.278,A -85,B 0,C 180,E1 -12216.888,E2 -12216.888} C_VEL
LIN {X 0,Y 375.983,Z 276.272,A -85,B 0,C 180,E1 -12220.34,E2 -12220.34} C_VEL
LIN {X 0,Y 376.014,Z 276.269,A -85,B 0,C 180,E1 -12223.719,E2 -12223.719} C_VEL
LIN {X 0,Y 376.089,Z 276.265,A -85,B 0,C 180,E1 -12227.043,E2 -12227.043} C_VEL
LIN {X 0,Y 376.105,Z 276.257,A -85,B 0,C 180,E1 -12230.319,E2 -12230.319} C_VEL
LIN {X 0,Y 376.224,Z 276.244,A -85,B 0,C 180,E1 -12233.566,E2 -12233.566} C_VEL
LIN {X 0,Y 376.341,Z 276.228,A -85,B 0,C 180,E1 -12237.86,E2 -12237.86} C_VEL
LIN {X 0,Y 376.476,Z 276.211,A -85,B 0,C 180,E1 -12240.001,E2 -12240.001} C_VEL
LIN {X 0,Y 376.171,Z 276.253,A -85,B 0,C 180,E1 -12243.214,E2 -12243.214} C_VEL
LIN {X 0,Y 376.232,Z 276.242,A -85,B 0,C 180,E1 -12246.436,E2 -12246.436} C_VEL
LIN {X 0,Y 376.193,Z 276.249,A -85,B 0,C 180,E1 -12248.596,E2 -12248.596} C_VEL
LIN {X 0,Y 376.038,Z 276.265,A -85,B 0,C 180,E1 -12251.865,E2 -12251.865} C_VEL
LIN {X 0,Y 376.047,Z 276.268,A -85,B 0,C 180,E1 -12255.169,E2 -12255.169} C_VEL
LIN {X 0,Y 375.998,Z 276.273,A -85,B 0,C 180,E1 -12258.528,E2 -12258.528} C_VEL
LIN {X 0,Y 375.947,Z 276.277,A -85,B 0,C 180,E1 -12261.956,E2 -12261.956} C_VEL
LIN {X 0,Y 375.995,Z 276.272,A -85,B 0,C 180,E1 -12265.462,E2 -12265.462} C_VEL
LIN {X 0,Y 375.961,Z 276.279,A -85,B 0,C 180,E1 -12269.081,E2 -12269.081} C_VEL
LIN {X 0,Y 375.94,Z 276.284,A -85,B 0,C 180,E1 -12272.83,E2 -12272.83} C_VEL
LIN {X 0,Y 375.949,Z 276.277,A -85,B 0,C 180,E1 -12275.417,E2 -12275.417} C_VEL
LIN {X 0,Y 375.964,Z 276.276,A -85,B 0,C 180,E1 -12278.272,E2 -12278.272} C_VEL
LIN {X 0,Y 375.926,Z 276.279,A -85,B 0,C 180,E1 -12281.602,E2 -12281.602} C_VEL
LIN {X 0,Y 375.92,Z 276.282,A -85,B 0,C 180,E1 -12285.27,E2 -12285.27} C_VEL
LIN {X 0,Y 375.928,Z 276.282,A -85,B 0,C 180,E1 -12288.401,E2 -12288.401} C_VEL
LIN {X 0,Y 375.968,Z 276.277,A -85,B 0,C 180,E1 -12291.731,E2 -12291.731} C_VEL
LIN {X 0,Y 375.976,Z 276.328,A -85,B 0,C 180,E1 -12293.568,E2 -12293.568} C_VEL
LIN {X 0,Y 379.82,Z 291.589,A -85,B 0,C 180,E1 -12296.667,E2 -12296.667} C_VEL
LIN {X 0,Y 383.65,Z 307.334,A -85,B 0,C 180,E1 -12299.715,E2 -12299.715} C_VEL
LIN {X 0,Y 383.58,Z 311.008,A -85,B 0,C 180,E1 -12300.352,E2 -12300.352} C_VEL
LIN {X 0,Y 383.237,Z 313.768,A -85,B 0,C 180,E1 -12300.812,E2 -12300.812} C_VEL
LIN {X 0,Y 389.631,Z 355.082,A -85,B 0,C 180,E1 -12302.3,E2 -12302.3} C_VEL
LIN {X 0,Y 385.346,Z 481.467,A -85,B 0,C 180,E1 -12305.308,E2 -12305.308} C_VEL
LIN {X 0,Y 384.427,Z 497.38,A -85,B 0,C 180,E1 -12305.892,E2 -12305.892} C_VEL
LIN {X 0,Y 383.349,Z 512.125,A -85,B 0,C 180,E1 -12306.636,E2 -12306.636} C_VEL
LIN {X 0,Y 382.173,Z 526.474,A -85,B 0,C 180,E1 -12307.57,E2 -12307.57} C_VEL
LIN {X 0,Y 380.862,Z 541.133,A -85,B 0,C 180,E1 -12308.77,E2 -12308.77} C_VEL
LIN {X 0,Y 379.529,Z 554.47,A -85,B 0,C 180,E1 -12310.109,E2 -12310.109} C_VEL
LIN {X 0,Y 378.33,Z 566.725,A -85,B 0,C 180,E1 -12311.593,E2 -12311.593} C_VEL
LIN {X 0,Y 377.258,Z 577.951,A -85,B 0,C 180,E1 -12313.218,E2 -12313.218} C_VEL
LIN {X 0,Y 376.368,Z 587.438,A -85,B 0,C 180,E1 -12314.847,E2 -12314.847} C_VEL
LIN {X 0,Y 375.67,Z 596.103,A -85,B 0,C 180,E1 -12316.61,E2 -12316.61} C_VEL
LIN {X 0,Y 375.189,Z 604.401,A -85,B 0,C 180,E1 -12318.658,E2 -12318.658} C_VEL
LIN {X 0,Y 374.786,Z 611.434,A -85,B 0,C 180,E1 -12320.83,E2 -12320.83} C_VEL
LIN {X 0,Y 374.688,Z 615.647,A -85,B 0,C 180,E1 -12322.457,E2 -12322.457} C_VEL
LIN {X 0,Y 374.673,Z 618.54,A -85,B 0,C 180,E1 -12323.806,E2 -12323.806} C_VEL
LIN {X 0,Y 374.578,Z 621.592,A -85,B 0,C 180,E1 -12325.697,E2 -12325.697} C_VEL
LIN {X 0,Y 374.715,Z 623.844,A -85,B 0,C 180,E1 -12327.852,E2 -12327.852} C_VEL
LIN {X 0,Y 374.654,Z 624.764,A -85,B 0,C 180,E1 -12330.001,E2 -12330.001} C_VEL
LIN {X 0,Y 374.692,Z 624.389,A -85,B 0,C 180,E1 -12332.151,E2 -12332.151} C_VEL
LIN {X 0,Y 374.574,Z 622.715,A -85,B 0,C 180,E1 -12334.306,E2 -12334.306} C_VEL
LIN {X 0,Y 374.575,Z 619.717,A -85,B 0,C 180,E1 -12336.465,E2 -12336.465} C_VEL
LIN {X 0,Y 374.718,Z 615.363,A -85,B 0,C 180,E1 -12338.631,E2 -12338.631} C_VEL
LIN {X 0,Y 375.035,Z 609.571,A -85,B 0,C 180,E1 -12340.802,E2 -12340.802} C_VEL
LIN {X 0,Y 375.659,Z 602.224,A -85,B 0,C 180,E1 -12342.975,E2 -12342.975} C_VEL
LIN {X 0,Y 376.615,Z 593.139,A -85,B 0,C 180,E1 -12345.146,E2 -12345.146} C_VEL
LIN {X 0,Y 377.782,Z 583.494,A -85,B 0,C 180,E1 -12347.039,E2 -12347.039} C_VEL
LIN {X 0,Y 379.23,Z 571.949,A -85,B 0,C 180,E1 -12348.929,E2 -12348.929} C_VEL
LIN {X 0,Y 380.855,Z 560.248,A -85,B 0,C 180,E1 -12350.526,E2 -12350.526} C_VEL
LIN {X 0,Y 382.8,Z 546.245,A -85,B 0,C 180,E1 -12352.11,E2 -12352.11} C_VEL
LIN {X 0,Y 384.64,Z 532.244,A -85,B 0,C 180,E1 -12353.417,E2 -12353.417} C_VEL
LIN {X 0,Y 386.53,Z 517.573,A -85,B 0,C 180,E1 -12354.534,E2 -12354.534} C_VEL
LIN {X 0,Y 388.441,Z 501.191,A -85,B 0,C 180,E1 -12355.522,E2 -12355.522} C_VEL
LIN {X 0,Y 390.219,Z 484.818,A -85,B 0,C 180,E1 -12356.257,E2 -12356.257} C_VEL
LIN {X 0,Y 391.497,Z 468.14,A -85,B 0,C 180,E1 -12356.811,E2 -12356.811} C_VEL
LIN {X 0,Y 396.167,Z 396.247,A -85,B 0,C 180,E1 -12358.855,E2 -12358.855} C_VEL
LIN {X 0,Y 399.199,Z 356.298,A -85,B 0,C 180,E1 -12360.059,E2 -12360.059} C_VEL
LIN {X 0,Y 398.164,Z 343.849,A -85,B 0,C 180,E1 -12360.739,E2 -12360.739} C_VEL
LIN {X 0,Y 396.045,Z 328.09,A -85,B 0,C 180,E1 -12361.794,E2 -12361.794} C_VEL
LIN {X 0,Y 394.86,Z 321.898,A -85,B 0,C 180,E1 -12362.299,E2 -12362.299} C_VEL
LIN {X 0,Y 391.197,Z 313.87,A -85,B 0,C 180,E1 -12363.399,E2 -12363.399} C_VEL
LIN {X 0,Y 388.248,Z 308.066,A -85,B 0,C 180,E1 -12364.348,E2 -12364.348} C_VEL
LIN {X 0,Y 385.033,Z 301.944,A -85,B 0,C 180,E1 -12365.544,E2 -12365.544} C_VEL
LIN {X 0,Y 383.232,Z 295.855,A -85,B 0,C 180,E1 -12367.948,E2 -12367.948} C_VEL
LIN {X 0,Y 381.801,Z 291.549,A -85,B 0,C 180,E1 -12370.112,E2 -12370.112} C_VEL
LIN {X 0,Y 380.538,Z 288.226,A -85,B 0,C 180,E1 -12372.375,E2 -12372.375} C_VEL
LIN {X 0,Y 379.761,Z 285.908,A -85,B 0,C 180,E1 -12374.689,E2 -12374.689} C_VEL
LIN {X 0,Y 379.272,Z 284.986,A -85,B 0,C 180,E1 -12376.715,E2 -12376.715} C_VEL
LIN {X 0,Y 379.235,Z 285.007,A -85,B 0,C 180,E1 -12379.562,E2 -12379.562} C_VEL
LIN {X 0,Y 379.534,Z 285.646,A -85,B 0,C 180,E1 -12381.055,E2 -12381.055} C_VEL
LIN {X 0,Y 380.276,Z 287.6,A -85,B 0,C 180,E1 -12383.244,E2 -12383.244} C_VEL
LIN {X 0,Y 383.339,Z 291.286,A -85,B 0,C 180,E1 -12384.54,E2 -12384.54} C_VEL
LIN {X 0,Y 384.725,Z 293.038,A -85,B 0,C 180,E1 -12385.058,E2 -12385.058} C_VEL
LIN {X 0,Y 388.033,Z 297.287,A -85,B 0,C 180,E1 -12386.189,E2 -12386.189} C_VEL
LIN {X 0,Y 391.462,Z 302.071,A -85,B 0,C 180,E1 -12387.237,E2 -12387.237} C_VEL
LIN {X 0,Y 395.354,Z 308.067,A -85,B 0,C 180,E1 -12388.325,E2 -12388.325} C_VEL
LIN {X 0,Y 399.969,Z 316.372,A -85,B 0,C 180,E1 -12389.523,E2 -12389.523} C_VEL
LIN {X 0,Y 401.369,Z 319.292,A -85,B 0,C 180,E1 -12389.875,E2 -12389.875} C_VEL
LIN {X 0,Y 395.204,Z 394.559,A -85,B 0,C 180,E1 -12392.136,E2 -12392.136} C_VEL
LIN {X 0,Y 391.869,Z 445.923,A -85,B 0,C 180,E1 -12393.653,E2 -12393.653} C_VEL
LIN {X 0,Y 390.615,Z 461.44,A -85,B 0,C 180,E1 -12394.31,E2 -12394.31} C_VEL
LIN {X 0,Y 389.151,Z 477.021,A -85,B 0,C 180,E1 -12395.201,E2 -12395.201} C_VEL
LIN {X 0,Y 387.722,Z 490.854,A -85,B 0,C 180,E1 -12396.214,E2 -12396.214} C_VEL
LIN {X 0,Y 386.113,Z 504.066,A -85,B 0,C 180,E1 -12397.386,E2 -12397.386} C_VEL
LIN {X 0,Y 384.323,Z 517.043,A -85,B 0,C 180,E1 -12398.776,E2 -12398.776} C_VEL
LIN {X 0,Y 382.707,Z 527.702,A -85,B 0,C 180,E1 -12400.139,E2 -12400.139} C_VEL
LIN {X 0,Y 381.15,Z 538.191,A -85,B 0,C 180,E1 -12401.731,E2 -12401.731} C_VEL
LIN {X 0,Y 379.636,Z 548.427,A -85,B 0,C 180,E1 -12403.601,E2 -12403.601} C_VEL
LIN {X 0,Y 378.212,Z 556.943,A -85,B 0,C 180,E1 -12405.471,E2 -12405.471} C_VEL
LIN {X 0,Y 377.103,Z 564.876,A -85,B 0,C 180,E1 -12407.623,E2 -12407.623} C_VEL
LIN {X 0,Y 376.205,Z 571.169,A -85,B 0,C 180,E1 -12409.777,E2 -12409.777} C_VEL
LIN {X 0,Y 375.614,Z 575.976,A -85,B 0,C 180,E1 -12411.932,E2 -12411.932} C_VEL
LIN {X 0,Y 375.242,Z 578.732,A -85,B 0,C 180,E1 -12413.547,E2 -12413.547} C_VEL
LIN {X 0,Y 375.015,Z 581.209,A -85,B 0,C 180,E1 -12415.7,E2 -12415.7} C_VEL
LIN {X 0,Y 374.814,Z 582.443,A -85,B 0,C 180,E1 -12417.85,E2 -12417.85} C_VEL
LIN {X 0,Y 374.659,Z 582.452,A -85,B 0,C 180,E1 -12419.999,E2 -12419.999} C_VEL
LIN {X 0,Y 374.771,Z 581.215,A -85,B 0,C 180,E1 -12422.149,E2 -12422.149} C_VEL
LIN {X 0,Y 374.752,Z 578.739,A -85,B 0,C 180,E1 -12424.301,E2 -12424.301} C_VEL
LIN {X 0,Y 374.949,Z 574.717,A -85,B 0,C 180,E1 -12426.566,E2 -12426.566} C_VEL
LIN {X 0,Y 375.216,Z 569.764,A -85,B 0,C 180,E1 -12428.617,E2 -12428.617} C_VEL
LIN {X 0,Y 375.675,Z 563.042,A -85,B 0,C 180,E1 -12430.781,E2 -12430.781} C_VEL
LIN {X 0,Y 376.392,Z 555.758,A -85,B 0,C 180,E1 -12432.673,E2 -12432.673} C_VEL
LIN {X 0,Y 377.074,Z 547.213,A -85,B 0,C 180,E1 -12434.517,E2 -12434.517} C_VEL
LIN {X 0,Y 377.974,Z 537.953,A -85,B 0,C 180,E1 -12436.194,E2 -12436.194} C_VEL
LIN {X 0,Y 379.002,Z 527.32,A -85,B 0,C 180,E1 -12437.815,E2 -12437.815} C_VEL
LIN {X 0,Y 380.118,Z 515.719,A -85,B 0,C 180,E1 -12439.302,E2 -12439.302} C_VEL
LIN {X 0,Y 381.399,Z 501.898,A -85,B 0,C 180,E1 -12440.775,E2 -12440.775} C_VEL
LIN {X 0,Y 382.596,Z 488.068,A -85,B 0,C 180,E1 -12441.978,E2 -12441.978} C_VEL
LIN {X 0,Y 383.75,Z 472.775,A -85,B 0,C 180,E1 -12443.044,E2 -12443.044} C_VEL
LIN {X 0,Y 384.682,Z 457.303,A -85,B 0,C 180,E1 -12443.883,E2 -12443.883} C_VEL
LIN {X 0,Y 385.421,Z 442.058,A -85,B 0,C 180,E1 -12444.494,E2 -12444.494} C_VEL
LIN {X 0,Y 386.071,Z 421.622,A -85,B 0,C 180,E1 -12445.038,E2 -12445.038} C_VEL
LIN {X 0,Y 389.906,Z 308.999,A -85,B 0,C 180,E1 -12447.689,E2 -12447.689} C_VEL
LIN {X 0,Y 383.477,Z 293.745,A -85,B 0,C 180,E1 -12448.484,E2 -12448.484} C_VEL
LIN {X 0,Y 376.042,Z 276.877,A -85,B 0,C 180,E1 -12449.43,E2 -12449.43} C_VEL
LIN {X 0,Y 375.952,Z 276.28,A -85,B 0,C 180,E1 -12449.482,E2 -12449.482} C_VEL
LIN {X 0,Y 375.95,Z 276.278,A -85,B 0,C 180,E1 -12452.827,E2 -12452.827} C_VEL
LIN {X 0,Y 375.957,Z 276.277,A -85,B 0,C 180,E1 -12455.414,E2 -12455.414} C_VEL
LIN {X 0,Y 375.938,Z 276.28,A -85,B 0,C 180,E1 -12458.262,E2 -12458.262} C_VEL
LIN {X 0,Y 375.922,Z 276.284,A -85,B 0,C 180,E1 -12461.597,E2 -12461.597} C_VEL
LIN {X 0,Y 375.925,Z 276.281,A -85,B 0,C 180,E1 -12465.267,E2 -12465.267} C_VEL
LIN {X 0,Y 375.932,Z 276.28,A -85,B 0,C 180,E1 -12468.398,E2 -12468.398} C_VEL
LIN {X 0,Y 375.97,Z 276.28,A -85,B 0,C 180,E1 -12471.728,E2 -12471.728} C_VEL
LIN {X 0,Y 375.977,Z 276.275,A -85,B 0,C 180,E1 -12475.331,E2 -12475.331} C_VEL
LIN {X 0,Y 375.954,Z 276.276,A -85,B 0,C 180,E1 -12478.436,E2 -12478.436} C_VEL
LIN {X 0,Y 375.931,Z 276.281,A -85,B 0,C 180,E1 -12482.135,E2 -12482.135} C_VEL
LIN {X 0,Y 375.973,Z 276.28,A -85,B 0,C 180,E1 -12485.716,E2 -12485.716} C_VEL
LIN {X 0,Y 375.993,Z 276.273,A -85,B 0,C 180,E1 -12489.196,E2 -12489.196} C_VEL
LIN {X 0,Y 376.027,Z 276.267,A -85,B 0,C 180,E1 -12492.599,E2 -12492.599} C_VEL
LIN {X 0,Y 376.083,Z 276.26,A -85,B 0,C 180,E1 -12496.341,E2 -12496.341} C_VEL
LIN {X 0,Y 376.112,Z 276.257,A -85,B 0,C 180,E1 -12500.317,E2 -12500.317} C_VEL
LIN {X 0,Y 376.222,Z 276.242,A -85,B 0,C 180,E1 -12502.485,E2 -12502.485} C_VEL
LIN {X 0,Y 376.161,Z 276.25,A -85,B 0,C 180,E1 -12504.638,E2 -12504.638} C_VEL
LIN {X 0,Y 376.342,Z 276.231,A -85,B 0,C 180,E1 -12507.858,E2 -12507.858} C_VEL
LIN {X 0,Y 376.48,Z 276.212,A -85,B 0,C 180,E1 -12509.999,E2 -12509.999} C_VEL
LIN {X 0,Y 376.176,Z 276.251,A -85,B 0,C 180,E1 -12513.212,E2 -12513.212} C_VEL
LIN {X 0,Y 376.235,Z 276.241,A -85,B 0,C 180,E1 -12516.434,E2 -12516.434} C_VEL
LIN {X 0,Y 376.196,Z 276.246,A -85,B 0,C 180,E1 -12518.594,E2 -12518.594} C_VEL
LIN {X 0,Y 376.04,Z 276.268,A -85,B 0,C 180,E1 -12521.862,E2 -12521.862} C_VEL
LIN {X 0,Y 376.047,Z 276.268,A -85,B 0,C 180,E1 -12525.166,E2 -12525.166} C_VEL
LIN {X 0,Y 376.013,Z 276.268,A -85,B 0,C 180,E1 -12526.413,E2 -12526.413} C_VEL
LIN {X 0,Y 375.335,Z 276.358,A -85,B 0,C 180,E1 -12527.307,E2 -12527.307} C_VEL
LIN {X 0,Y 372.48,Z 276.709,A -85,B 0,C 180,E1 -12528.759,E2 -12528.759} C_VEL
LIN {X 0,Y 370.061,Z 277.012,A -85,B 0,C 180,E1 -12529.933,E2 -12529.933} C_VEL
LIN {X 0,Y 369.012,Z 277.142,A -85,B 0,C 180,E1 -12530.841,E2 -12530.841} C_VEL
LIN {X 0,Y 368.921,Z 277.155,A -85,B 0,C 180,E1 -12531.149,E2 -12531.149} C_VEL
LIN {X 0,Y 368.945,Z 277.15,A -85,B 0,C 180,E1 -12534.774,E2 -12534.774} C_VEL
LIN {X 0,Y 368.95,Z 277.153,A -85,B 0,C 180,E1 -12537.202,E2 -12537.202} C_VEL
LIN {X 0,Y 368.916,Z 277.155,A -85,B 0,C 180,E1 -12540.953,E2 -12540.953} C_VEL
LIN {X 0,Y 368.916,Z 277.155,A -85,B 0,C 180,E1 -12545.001,E2 -12545.001} C_VEL
LIN {X 0,Y 368.896,Z 277.156,A -85,B 0,C 180,E1 -12548.64,E2 -12548.64} C_VEL
LIN {X 0,Y 368.868,Z 277.159,A -85,B 0,C 180,E1 -12552.009,E2 -12552.009} C_VEL
LIN {X 0,Y 368.894,Z 277.161,A -85,B 0,C 180,E1 -12555.18,E2 -12555.18} C_VEL
LIN {X 0,Y 368.868,Z 277.158,A -85,B 0,C 180,E1 -12558.177,E2 -12558.177} C_VEL
LIN {X 0,Y 368.894,Z 277.161,A -85,B 0,C 180,E1 -12561.359,E2 -12561.359} C_VEL
LIN {X 0,Y 368.922,Z 277.158,A -85,B 0,C 180,E1 -12565.146,E2 -12565.146} C_VEL
LIN {X 0,Y 368.915,Z 277.158,A -85,B 0,C 180,E1 -12569.046,E2 -12569.046} C_VEL
LIN {X 0,Y 368.961,Z 277.15,A -85,B 0,C 180,E1 -12571.564,E2 -12571.564} C_VEL
LIN {X 0,Y 368.985,Z 277.144,A -85,B 0,C 180,E1 -12574.02,E2 -12574.02} C_VEL
LIN {X 0,Y 368.91,Z 277.155,A -85,B 0,C 180,E1 -12577.605,E2 -12577.605} C_VEL
LIN {X 0,Y 368.944,Z 277.156,A -85,B 0,C 180,E1 -12581.106,E2 -12581.106} C_VEL
LIN {X 0,Y 368.983,Z 277.145,A -85,B 0,C 180,E1 -12584.536,E2 -12584.536} C_VEL
LIN {X 0,Y 368.991,Z 277.143,A -85,B 0,C 180,E1 -12587.907,E2 -12587.907} C_VEL
LIN {X 0,Y 369.173,Z 277.121,A -85,B 0,C 180,E1 -12591.847,E2 -12591.847} C_VEL
LIN {X 0,Y 369.127,Z 277.128,A -85,B 0,C 180,E1 -12594.538,E2 -12594.538} C_VEL
LIN {X 0,Y 369.306,Z 277.104,A -85,B 0,C 180,E1 -12597.82,E2 -12597.82} C_VEL
LIN {X 0,Y 369.445,Z 277.086,A -85,B 0,C 180,E1 -12600.001,E2 -12600.001} C_VEL
LIN {X 0,Y 369.303,Z 277.104,A -85,B 0,C 180,E1 -12602.182,E2 -12602.182} C_VEL
LIN {X 0,Y 369.194,Z 277.12,A -85,B 0,C 180,E1 -12606.559,E2 -12606.559} C_VEL
LIN {X 0,Y 369.126,Z 277.131,A -85,B 0,C 180,E1 -12608.762,E2 -12608.762} C_VEL
LIN {X 0,Y 368.993,Z 277.143,A -85,B 0,C 180,E1 -12612.094,E2 -12612.094} C_VEL
LIN {X 0,Y 368.986,Z 277.145,A -85,B 0,C 180,E1 -12615.466,E2 -12615.466} C_VEL
LIN {X 0,Y 368.947,Z 277.155,A -85,B 0,C 180,E1 -12618.895,E2 -12618.895} C_VEL
LIN {X 0,Y 368.914,Z 277.154,A -85,B 0,C 180,E1 -12622.397,E2 -12622.397} C_VEL
LIN {X 0,Y 368.99,Z 277.143,A -85,B 0,C 180,E1 -12625.982,E2 -12625.982} C_VEL
LIN {X 0,Y 368.95,Z 277.155,A -85,B 0,C 180,E1 -12628.812,E2 -12628.812} C_VEL
LIN {X 0,Y 368.889,Z 277.157,A -85,B 0,C 180,E1 -12632.24,E2 -12632.24} C_VEL
LIN {X 0,Y 368.92,Z 277.156,A -85,B 0,C 180,E1 -12635.003,E2 -12635.003} C_VEL
LIN {X 0,Y 368.899,Z 277.16,A -85,B 0,C 180,E1 -12638.642,E2 -12638.642} C_VEL
LIN {X 0,Y 368.873,Z 277.158,A -85,B 0,C 180,E1 -12642.011,E2 -12642.011} C_VEL
LIN {X 0,Y 368.877,Z 277.16,A -85,B 0,C 180,E1 -12645.178,E2 -12645.178} C_VEL
LIN {X 0,Y 368.877,Z 277.159,A -85,B 0,C 180,E1 -12648.179,E2 -12648.179} C_VEL
LIN {X 0,Y 368.903,Z 277.158,A -85,B 0,C 180,E1 -12651.362,E2 -12651.362} C_VEL
LIN {X 0,Y 368.947,Z 277.325,A -85,B 0,C 180,E1 -12653.193,E2 -12653.193} C_VEL
LIN {X 0,Y 372.902,Z 292.882,A -85,B 0,C 180,E1 -12656.419,E2 -12656.419} C_VEL
LIN {X 0,Y 376.563,Z 308.15,A -85,B 0,C 180,E1 -12659.429,E2 -12659.429} C_VEL
LIN {X 0,Y 376.904,Z 309.969,A -85,B 0,C 180,E1 -12659.773,E2 -12659.773} C_VEL
LIN {X 0,Y 376.516,Z 313.51,A -85,B 0,C 180,E1 -12660.378,E2 -12660.378} C_VEL
LIN {X 0,Y 383.033,Z 355.656,A -85,B 0,C 180,E1 -12661.927,E2 -12661.927} C_VEL
LIN {X 0,Y 378.549,Z 480.751,A -85,B 0,C 180,E1 -12664.981,E2 -12664.981} C_VEL
LIN {X 0,Y 377.624,Z 496.72,A -85,B 0,C 180,E1 -12665.576,E2 -12665.576} C_VEL
LIN {X 0,Y 376.535,Z 511.686,A -85,B 0,C 180,E1 -12666.345,E2 -12666.345} C_VEL
LIN {X 0,Y 375.327,Z 525.891,A -85,B 0,C 180,E1 -12667.283,E2 -12667.283} C_VEL
LIN {X 0,Y 373.964,Z 540.577,A -85,B 0,C 180,E1 -12668.504,E2 -12668.504} C_VEL
LIN {X 0,Y 372.607,Z 553.948,A -85,B 0,C 180,E1 -12669.867,E2 -12669.867} C_VEL
LIN {X 0,Y 371.353,Z 566.226,A -85,B 0,C 180,E1 -12671.377,E2 -12671.377} C_VEL
LIN {X 0,Y 370.345,Z 576.633,A -85,B 0,C 180,E1 -12672.896,E2 -12672.896} C_VEL
LIN {X 0,Y 369.42,Z 586.283,A -85,B 0,C 180,E1 -12674.555,E2 -12674.555} C_VEL
LIN {X 0,Y 368.626,Z 595.689,A -85,B 0,C 180,E1 -12676.493,E2 -12676.493} C_VEL
LIN {X 0,Y 368.128,Z 603.499,A -85,B 0,C 180,E1 -12678.438,E2 -12678.438} C_VEL
LIN {X 0,Y 367.733,Z 610.656,A -85,B 0,C 180,E1 -12680.653,E2 -12680.653} C_VEL
LIN {X 0,Y 367.575,Z 616.194,A -85,B 0,C 180,E1 -12682.862,E2 -12682.862} C_VEL
LIN {X 0,Y 367.559,Z 619.336,A -85,B 0,C 180,E1 -12684.515,E2 -12684.515} C_VEL
LIN {X 0,Y 367.523,Z 622.327,A -85,B 0,C 180,E1 -12686.713,E2 -12686.713} C_VEL
LIN {X 0,Y 367.649,Z 623.326,A -85,B 0,C 180,E1 -12687.81,E2 -12687.81} C_VEL
LIN {X 0,Y 367.586,Z 624.314,A -85,B 0,C 180,E1 -12690.001,E2 -12690.001} C_VEL
LIN {X 0,Y 367.591,Z 624.001,A -85,B 0,C 180,E1 -12692.193,E2 -12692.193} C_VEL
LIN {X 0,Y 367.499,Z 622.371,A -85,B 0,C 180,E1 -12694.389,E2 -12694.389} C_VEL
LIN {X 0,Y 367.493,Z 619.413,A -85,B 0,C 180,E1 -12696.59,E2 -12696.59} C_VEL
LIN {X 0,Y 367.633,Z 615.119,A -85,B 0,C 180,E1 -12698.798,E2 -12698.798} C_VEL
LIN {X 0,Y 368.017,Z 609.393,A -85,B 0,C 180,E1 -12701.011,E2 -12701.011} C_VEL
LIN {X 0,Y 368.666,Z 602.127,A -85,B 0,C 180,E1 -12703.225,E2 -12703.225} C_VEL
LIN {X 0,Y 369.545,Z 594.343,A -85,B 0,C 180,E1 -12705.16,E2 -12705.16} C_VEL
LIN {X 0,Y 370.741,Z 585.041,A -85,B 0,C 180,E1 -12707.089,E2 -12707.089} C_VEL
LIN {X 0,Y 372.191,Z 574.25,A -85,B 0,C 180,E1 -12708.964,E2 -12708.964} C_VEL
LIN {X 0,Y 374.079,Z 561.705,A -85,B 0,C 180,E1 -12710.771,E2 -12710.771} C_VEL
LIN {X 0,Y 376.067,Z 548.223,A -85,B 0,C 180,E1 -12712.383,E2 -12712.383} C_VEL
LIN {X 0,Y 378.229,Z 533.354,A -85,B 0,C 180,E1 -12713.839,E2 -12713.839} C_VEL
LIN {X 0,Y 380.357,Z 517.932,A -85,B 0,C 180,E1 -12715.053,E2 -12715.053} C_VEL
LIN {X 0,Y 382.469,Z 501.141,A -85,B 0,C 180,E1 -12716.096,E2 -12716.096} C_VEL
LIN {X 0,Y 384.403,Z 484.449,A -85,B 0,C 180,E1 -12716.869,E2 -12716.869} C_VEL
LIN {X 0,Y 385.818,Z 467.231,A -85,B 0,C 180,E1 -12717.459,E2 -12717.459} C_VEL
LIN {X 0,Y 390.837,Z 396.769,A -85,B 0,C 180,E1 -12719.532,E2 -12719.532} C_VEL
LIN {X 0,Y 394.092,Z 357.874,A -85,B 0,C 180,E1 -12720.735,E2 -12720.735} C_VEL
LIN {X 0,Y 393.233,Z 345.937,A -85,B 0,C 180,E1 -12721.414,E2 -12721.414} C_VEL
LIN {X 0,Y 391.264,Z 329.93,A -85,B 0,C 180,E1 -12722.536,E2 -12722.536} C_VEL
LIN {X 0,Y 390.502,Z 325.88,A -85,B 0,C 180,E1 -12722.89,E2 -12722.89} C_VEL
LIN {X 0,Y 387.254,Z 318.562,A -85,B 0,C 180,E1 -12723.947,E2 -12723.947} C_VEL
LIN {X 0,Y 384.73,Z 313.362,A -85,B 0,C 180,E1 -12724.825,E2 -12724.825} C_VEL
LIN {X 0,Y 381.348,Z 307.03,A -85,B 0,C 180,E1 -12726.115,E2 -12726.115} C_VEL
LIN {X 0,Y 377.431,Z 300.081,A -85,B 0,C 180,E1 -12727.916,E2 -12727.916} C_VEL
LIN {X 0,Y 376.153,Z 295.95,A -85,B 0,C 180,E1 -12730,E2 -12730} C_VEL
LIN {X 0,Y 374.839,Z 292.408,A -85,B 0,C 180,E1 -12732.454,E2 -12732.454} C_VEL
LIN {X 0,Y 374.197,Z 290.367,A -85,B 0,C 180,E1 -12734.463,E2 -12734.463} C_VEL
LIN {X 0,Y 373.536,Z 289.158,A -85,B 0,C 180,E1 -12737.364,E2 -12737.364} C_VEL
LIN {X 0,Y 373.658,Z 289.541,A -85,B 0,C 180,E1 -12740.245,E2 -12740.245} C_VEL
LIN {X 0,Y 373.928,Z 289.954,A -85,B 0,C 180,E1 -12740.778,E2 -12740.778} C_VEL
LIN {X 0,Y 377.524,Z 293.734,A -85,B 0,C 180,E1 -12742.829,E2 -12742.829} C_VEL
LIN {X 0,Y 381.781,Z 298.936,A -85,B 0,C 180,E1 -12744.673,E2 -12744.673} C_VEL
LIN {X 0,Y 385.2,Z 303.579,A -85,B 0,C 180,E1 -12745.912,E2 -12745.912} C_VEL
LIN {X 0,Y 388.285,Z 308.006,A -85,B 0,C 180,E1 -12746.906,E2 -12746.906} C_VEL
LIN {X 0,Y 393.034,Z 315.797,A -85,B 0,C 180,E1 -12748.299,E2 -12748.299} C_VEL
LIN {X 0,Y 396.321,Z 322.267,A -85,B 0,C 180,E1 -12749.2,E2 -12749.2} C_VEL
LIN {X 0,Y 389.504,Z 399.118,A -85,B 0,C 180,E1 -12751.582,E2 -12751.582} C_VEL
LIN {X 0,Y 386.193,Z 446.314,A -85,B 0,C 180,E1 -12753.022,E2 -12753.022} C_VEL
LIN {X 0,Y 384.914,Z 461.497,A -85,B 0,C 180,E1 -12753.681,E2 -12753.681} C_VEL
LIN {X 0,Y 383.279,Z 477.608,A -85,B 0,C 180,E1 -12754.62,E2 -12754.62} C_VEL
LIN {X 0,Y 381.683,Z 491.684,A -85,B 0,C 180,E1 -12755.669,E2 -12755.669} C_VEL
LIN {X 0,Y 379.964,Z 504.761,A -85,B 0,C 180,E1 -12756.855,E2 -12756.855} C_VEL
LIN {X 0,Y 378.032,Z 517.951,A -85,B 0,C 180,E1 -12758.301,E2 -12758.301} C_VEL
LIN {X 0,Y 376.194,Z 529.2,A -85,B 0,C 180,E1 -12759.78,E2 -12759.78} C_VEL
LIN {X 0,Y 374.549,Z 539.501,A -85,B 0,C 180,E1 -12761.398,E2 -12761.398} C_VEL
LIN {X 0,Y 372.918,Z 549.585,A -85,B 0,C 180,E1 -12763.297,E2 -12763.297} C_VEL
LIN {X 0,Y 371.41,Z 557.972,A -85,B 0,C 180,E1 -12765.199,E2 -12765.199} C_VEL
LIN {X 0,Y 370.218,Z 565.788,A -85,B 0,C 180,E1 -12767.39,E2 -12767.39} C_VEL
LIN {X 0,Y 369.255,Z 571.983,A -85,B 0,C 180,E1 -12769.582,E2 -12769.582} C_VEL
LIN {X 0,Y 368.607,Z 576.693,A -85,B 0,C 180,E1 -12771.778,E2 -12771.778} C_VEL
LIN {X 0,Y 368.218,Z 579.376,A -85,B 0,C 180,E1 -12773.423,E2 -12773.423} C_VEL
LIN {X 0,Y 367.953,Z 581.791,A -85,B 0,C 180,E1 -12775.617,E2 -12775.617} C_VEL
LIN {X 0,Y 367.753,Z 582.947,A -85,B 0,C 180,E1 -12777.809,E2 -12777.809} C_VEL
LIN {X 0,Y 367.591,Z 582.867,A -85,B 0,C 180,E1 -12779.999,E2 -12779.999} C_VEL
LIN {X 0,Y 367.689,Z 581.542,A -85,B 0,C 180,E1 -12782.19,E2 -12782.19} C_VEL
LIN {X 0,Y 367.679,Z 578.971,A -85,B 0,C 180,E1 -12784.384,E2 -12784.384} C_VEL
LIN {X 0,Y 367.885,Z 575.08,A -85,B 0,C 180,E1 -12786.581,E2 -12786.581} C_VEL
LIN {X 0,Y 368.171,Z 569.782,A -85,B 0,C 180,E1 -12788.783,E2 -12788.783} C_VEL
LIN {X 0,Y 368.64,Z 562.936,A -85,B 0,C 180,E1 -12790.99,E2 -12790.99} C_VEL
LIN {X 0,Y 369.4,Z 555.517,A -85,B 0,C 180,E1 -12792.917,E2 -12792.917} C_VEL
LIN {X 0,Y 370.141,Z 546.535,A -85,B 0,C 180,E1 -12794.851,E2 -12794.851} C_VEL
LIN {X 0,Y 371.249,Z 535.698,A -85,B 0,C 180,E1 -12796.779,E2 -12796.779} C_VEL
